# B&R Automation Studio project perfxxl (part 3)

#### sram.c
```c
#ifdef _DEFAULT_INCLUDES
	#include <AsDefault.h>
#endif
/****************************************************************************/
/*	Zugriff auf remanenten Speicher*/
/*																			*/
/*																			*/
/*	Versionsgeschichte:														*/
/*  Version		Datum		Änderung										von		*/
/*	1.00		16.09.02	erste Implementation								HA		*/
/*	1.10		31.03.03	bei Änderung Aufl. und Speed speichern		HA		*/
/*	1.11		20.05.03	floats auf Gültigkeit prüfen				HA		*/
/*																			*/
/****************************************************************************/

#include <bur/plc.h>
#include <bur/plctypes.h>
#include <math.h>
#include <asstring.h>
#include "glob_var.h"
#include "egmglob_var.h"
#include <fileio.h>

#define	MAXFILELIST	32
#define MAXFILES	50
#define MAXFILENAMELENGTH	32

#define OVERALLSRAMSIZEWORDS 12500
#define OVERALLSRAMSIZEEBYTES 25000

typedef struct{
BOOL enable;
UDINT len;
UDINT offset;
UDINT	address;
}puttyp;
typedef struct{
BOOL enable;
UDINT len;
UDINT offset;
UDINT	address;
}gettyp;
puttyp put;
gettyp get;

_LOCAL UINT             wStatus, wError;
_LOCAL UDINT            dwDirNum, dwFileNum, dwCounter;
_LOCAL DirInfo_typ      DInfo;
_LOCAL DirCreate_typ      DCreate;
_LOCAL BOOL Created;
_GLOBAL BOOL PreheatParamEnter,DeveloperTankParamEnter;

_LOCAL STRING targetstring[20];
int i,j;
USINT tmp[OVERALLSRAMSIZEEBYTES];
_GLOBAL USINT *TmpPtr;

int len;
_GLOBAL UDINT	PlatesMade;
_GLOBAL	BOOL	savePlatesMade;
		BOOL	loadPlatesMade;
_GLOBAL	STRING FileIOName[MAXFILENAMELENGTH];
_GLOBAL	STRING	FileType[5];
_GLOBAL	UDINT *FileIOData;
_GLOBAL	UDINT	FileIOLength;
_GLOBAL	BOOL	WriteFileCmd,ReadFileCmd,DeleteFileCmd,WriteFileOK,ReadFileOK,DeleteFileOK,
				FileNotExisting,ReadDirCmd,ReadDirOK,NoDisk;
_GLOBAL	BOOL ParameterChanged;

_LOCAL	BOOL	StartUp,ReadActive,WriteActive,SaveToFile;
_LOCAL	BOOL	ClearSRAM,LoadSRAMFromFile;
_GLOBAL BOOL	PutTmpDataToSRAM,GetTmpDataFromSRAM;
BOOL	DontResetMotorData;
_GLOBAL BOOL MirroredMachine;

_GLOBAL SINT SRAM[OVERALLSRAMSIZEEBYTES]	_VAR_RETAIN;
_GLOBAL BOOL	EGMsaveParameterData;
_LOCAL INT	Test1,Test2,Test3;

_LOCAL	STRING	MagicNumber[10];
_GLOBAL	DATE_AND_TIME	OffTime,OnTime;

void SRAMPut(puttyp *param)
{
	memcpy(&SRAM[0]+param->offset*2,(SINT *)(param->address),param->len *2);
}

void SRAMGet(gettyp *param)
{
	memcpy((SINT *)(param->address),&SRAM[0]+param->offset*2,param->len *2);
}

void InitXData(void)
{
	ClearSRAM = 0;
	X_Param.RefSpeed1		= 20;
	X_Param.RefSpeed2		= 10;
	X_Param.RefSpeed3		= 5;
	X_Param.ManSpeed1		= 20;
	X_Param.ManSpeed2		= 50;
	X_Param.ParkSpeed		= 195;
/*Positionen*/
	X_Param.Offset			= 0;		/*Nullpunktkorrektur*/
	X_Param.ParkPosition	= -3.0;
	X_Param.InkrementeProMm	= 2730.666;
	X_Param.MinPosition	= -37.0;
	X_Param.MaxPosition	= 1258.0;
}

void InitGlobalData(void)
{
	PlatesMade = 0;

	PlateParameter.XOffset = 0.0;
	PlateParameter.YOffset = 0.0;
	PlateParameter.Length  = 320.0;
	PlateParameter.Width   = 600.0;
	PlateParameter.Thickness = 0.30;
	PlateParameter.Sensitivity = 100.0;

	strcpy(GlobalParameter.MachineName,"LS Performance XXL");
	strcpy(GlobalParameter.MachineNumber,"12345");
	strcpy(GlobalParameter.CustomerName,"eintragen!!");
	GlobalParameter.ScansPerMinute			= 96000;
	GlobalParameter.Resolution				= 1270;
	GlobalParameter.MaxPlateLength			= 1250; /*not in use*/
	GlobalParameter.MinPlateLength			= 250;  /*not in use*/
	GlobalParameter.TrolleyRightOffset		= 73650;/*not in use*/
	GlobalParameter.AlternatingTrolleys		= FALSE;/*not in use*/
	GlobalParameter.XSimulation				= FALSE;
	GlobalParameter.TBSimulation			= FALSE;
	GlobalParameter.ProcessorSimulation		= FALSE;
	GlobalParameter.PunchSimulation			= FALSE;
	GlobalParameter.PaperRemoveEnabled		= TRUE;
	GlobalParameter.UseOldTiffBlaster		= FALSE;/*not in use*/
	GlobalParameter.Dummy					= FALSE;
	GlobalParameter.Language				= 1;
	GlobalParameter.DeloaderTurnStation		= 0;
	GlobalParameter.FlexibleFeeder			= 0;
	GlobalParameter.AutomaticTrolleyOpenClose	= TRUE;
	GlobalParameter.TrolleyLeft				= 0;
	GlobalParameter.TrolleyRight			= 0;
	GlobalParameter.RealLaserPower			= 300;
	GlobalParameter.LaserPower = (GlobalParameter.RealLaserPower+5) / 10;
	GlobalParameter.MirroredMachine			= 0; /* !=42: not mirrored; 42: mirrored*/
	GlobalParameter.SlowModeWaitTime		= 2000; /* 20 sec default */
	GlobalParameter.DisableSlowMode			= 1;

	Expose_Param.ScansPerMinute			= 96000;
	Expose_Param.Resolution				= 1270;

/*TROLLEYS*/
	for(i = 0; i < MAXTROLLEYS; i++)
	{
		strcpy( Trolleys[i].Name,"Trolley");
		Trolleys[i].Number 				= i;	/*bugfix i instead of i+1*/
		Trolleys[i].PlateType 			= 1;
		Trolleys[i].Empty 				= FALSE;
		Trolleys[i].Single 				= FALSE;
		Trolleys[i].Double 				= TRUE;
		Trolleys[i].NoCover		 		= FALSE;
		Trolleys[i].LeftStack 			= TRUE;
		Trolleys[i].RightStack 			= FALSE;
		Trolleys[i].PlatesLeft 			= 0;
		Trolleys[i].PlatesRight 		= 0;
		Trolleys[i].OpenStart 			= 175600;
		Trolleys[i].OpenStop 			= 353100;
		Trolleys[i].CloseStart 			= 353100;
		Trolleys[i].CloseStop 			= 174440;
		Trolleys[i].TakePlateLeft 		= 8300;  /* not in use*/
		Trolleys[i].TakePlateRight 		= 57000; /* not in use*/
		Trolleys[i].TakePaperLeft 		= 335000;
		Trolleys[i].TakePaperRight 		= 335000;
		Trolleys[i].EmptyLeft 			= FALSE;
		Trolleys[i].EmptyRight 			= FALSE;
		Trolleys[i].EmptyPositions[0] 			= 64000;
		Trolleys[i].EmptyPositions[1] 			= 64000;
		Trolleys[i].EmptyPositions[2] 			= 64000;
	}

/*PLATETYPES*/
	for(i = 0; i < MAXPLATETYPES; i++)
	{
		strcpy( PlateTypes[i].Name,"Platte");
		PlateTypes[i].Number 				= i; /*bugfix i instead of i+1*/
		PlateTypes[i].Length 				= 312.00;
		PlateTypes[i].XOffset 				= 0.00;
		PlateTypes[i].Width 				= 600.00;
		PlateTypes[i].YOffset 				= 10.00;
		PlateTypes[i].Thickness 				= 0.32;
		PlateTypes[i].TakePlatePosition 				= 100000;
		PlateTypes[i].ReleasePlatePosition 			= 10000;
		PlateTypes[i].ReleasePlatePosition2 			= 10000;
		PlateTypes[i].TurnMode							= 0;
		PlateTypes[i].SeparateBeltTracks	= 0;
	}

/*FEEDER*/
	FeederParameter.HorizontalPositions.ReleasePlate 				= 500;/* not in use*/
	FeederParameter.HorizontalPositions.TakePlate 				= 1500;/* not in use*/
	FeederParameter.VerticalPositions.Up 							= 2000;
	FeederParameter.VerticalPositions.EnablePaperRemove 		= 22000;
	FeederParameter.VerticalPositions.AboveTrolley 				= 22000;
	FeederParameter.VerticalPositions.MaxDown	 				= 70000;
	FeederParameter.VerticalPositions.PreRelease 					= 2000;
	FeederParameter.VerticalPositions.ReleasePlate 				= 2000;
	FeederParameter.VerticalPositions.SpeedChangePosition 		= 18200;
	FeederParameter.VacuumOnTime								= 100;
	FeederParameter.VacuumOffTime								= 50;
	FeederParameter.SpeedUpSlow									= 700;
	FeederParameter.SpeedUpFast									= 7000;
	FeederParameter.Stack0Pos									= -186000;/* not in use*/
	FeederParameter.Stack20Pos									= -183248;/* not in use*/
	FeederParameter.SlowDownPos									= 1000;
	FeederParameter.StackDetectSpeed							= 500;
	FeederParameter.PanoramaAdapter							= 25000;
	FeederParameter.SuckRepitions								= 0;
	FeederParameter.ShakeRepitions								= 0;
	FeederParameter.ShakeTime									= 30;
	FeederParameter.ShakeWay									= 3000;
	FeederParameter.WaitForExposer								= 0;
	FeederParameter.IgnoreVacuumSwitch							= 0;
	FeederParameter.HorPositionPano							= 2000;
	FeederParameter.MaxTablePosition							= 170.0;
	FeederParameter.MinTablePosDrop							= 1180.0;
	FeederParameter.DropOffset									= 20.0;/* not in use */

/* Paper Remove */
	PaperRemoveParameter.HorizontalPositions.EnableFeeder 			= 126000;
	PaperRemoveParameter.HorizontalPositions.PaperReleaseSingle		= 70000;
	PaperRemoveParameter.HorizontalPositions.PaperReleasePanorama	= 50000;

/*folgende Werte werden im Ablauf errechnet*/
	PaperRemoveParameter.HorizontalPositions.PaperRemoveLeft		= -120000;
	PaperRemoveParameter.HorizontalPositions.PaperRemoveRight		= -196000;
	PaperRemoveParameter.HorizontalPositions.TrolleyCloseRightStart	= -196000;
	PaperRemoveParameter.HorizontalPositions.TrolleyCloseRightStop	= -178000;
	PaperRemoveParameter.HorizontalPositions.TrolleyOpenRightStart	= -178000;
	PaperRemoveParameter.HorizontalPositions.TrolleyOpenRightStop	= -196000;
	PaperRemoveParameter.HorizontalPositions.PaletteDetectStartPos	=  120000;
	PaperRemoveParameter.HorizontalPositions.PaletteDetectEndPos	=  130000;
	PaperRemoveParameter.HorizontalPositions.TrolleyOpenRightStop	= -196000;
/* bis hier*/
	PaperRemoveParameter.VerticalPositions.Up						= 300;
	PaperRemoveParameter.VerticalPositions.Down						= 13000;
	PaperRemoveParameter.VerticalPositions.OnTrolley				= 1200;
	PaperRemoveParameter.TrolleyOpenCloseSpeed						= 1000;
	PaperRemoveParameter.PaperRemoveSpeed							= 5000;
	PaperRemoveParameter.TrolleyDetectSpeed							= 500;
	PaperRemoveParameter.TrolleyOpenDownSpeed						= 300;
	PaperRemoveParameter.TrolleyOpenUpSpeed							= 800;
	PaperRemoveParameter.PaperRemoveDownSpeed						= 1000;
	PaperRemoveParameter.PaperRemoveUpSpeed							= 1500;
	PaperRemoveParameter.TrolleyDetectStartPos						= 180000;
	PaperRemoveParameter.TrolleyDetectEndPos						= 280000;
	PaperRemoveParameter.MaxCurrentDown								= 2000;
	PaperRemoveParameter.MaxCurrentUp								= 5000;
	PaperRemoveParameter.GripOnTime									= 100;
	PaperRemoveParameter.GripOffTime								= 80;
	PaperRemoveParameter.TimeoutOnTrolley							= 100;
	PaperRemoveParameter.PaletteDetectSpeed							= 300;
	PaperRemoveParameter.TimeoutUpFromTrolley						= 100;
	PaperRemoveParameter.TimeoutOpenTrolleySmall					= 1000;/* not in use*/
	PaperRemoveParameter.TimeoutOpenTrolleyBig						= 2000;/* not in use*/
	PaperRemoveParameter.PaperGripCycles							= 0;
	PaperRemoveParameter.HorPositionPano							= 300000;
	PaperRemoveParameter.PaperReleasePosVertical					= 10000;

/*Adjuster*/
	AdjusterParameter.PinsUpTime									= 20;
	AdjusterParameter.PinsDownTime									= 20;
	AdjusterParameter.TableVacuumOnDelay							= 10;
	AdjusterParameter.TableVacuumOffDelay							= 20;
	AdjusterParameter.AdjVacuumOnDelay							= 50;
	AdjusterParameter.AdjVacuumOffDelay							= 10;
	AdjusterParameter.BlowairOnDelay								= 10;
	AdjusterParameter.BlowairOffDelay								= 10;
	AdjusterParameter.TimeoutAdjustedPosition						= 100;
	AdjusterParameter.MaxFailedPlates								= 0;
	AdjusterParameter.AddBlowairValveDelay						    = 1;
	AdjusterParameter.MaxAttempts									= 3;
	AdjusterParameter.AdjActiveTime									= 30;
	AdjusterParameter.AdjInactiveTime								= 30;
	AdjusterParameter.AdjustSim										= FALSE;
	AdjusterParameter.FeederAdjustposition							= 6450;
	AdjusterParameter.FeederFixposition							    = 7500;

/*DELOADER*/
	DeloaderParameter.MaxPlateTakePosition							= 100000;
	DeloaderParameter.PlateReleasePosition							= 10000;
	DeloaderParameter.PlateReleasePosition2							= 10000;
	DeloaderParameter.TurnEnabledPosition							= 50000;
	DeloaderParameter.MinTablePositionTake							= 235.0;
	DeloaderParameter.MaxTablePositionRelease						= 500.0;
	DeloaderParameter.Turn0Position									= 15400;
	DeloaderParameter.Turn90Position								= 26100;
	DeloaderParameter.Turn180Position								= 36800;
	DeloaderParameter.ConveyorBeltSpeed								= 300;
	DeloaderParameter.TableDeloadSpeedManual								= 200.0;
	DeloaderParameter.TableDeloadSpeed								= 200.0;
	DeloaderParameter.TurnSpeed										= 2000;
	DeloaderParameter.VacuumOnTime									= 50;
	DeloaderParameter.VacuumOffTime									= 50;
	DeloaderParameter.PlateLengthAddition								= 120;
	DeloaderParameter.ConveyorBeltDelay								= 500;
	DeloaderParameter.EGMStopDelay									= 4500;
	DeloaderParameter.ShiftedLayingOff								= 0;
	DeloaderParameter.PinsUpDelay									= 200;
	DeloaderParameter.PinsDownDelay								= 200;
	DeloaderParameter.EnableStopPins								= 0;
	DeloaderParameter.SeparateSensors								= 0;
	DeloaderParameter.StartTablePosition                           = -6.0;
	DeloaderParameter.EndTablePosition                             = 1258;
	DeloaderParameter.ConvLateralMoveTime                          = 200;
	DeloaderParameter.ConvLateralPulseTime                          = 30;

	for (i=1;i<MAXLASERPOWERSETTINGS;i++)
	{
		LaserPowerSettings[i].Resolution = 0;
		for (j = 1;j<MAXPLATETYPES;j++)
			LaserPowerSettings[i].LaserPower[j] = 0;
	}
}

void InitMotorData(void)
{
	Motors[FEEDER_VERTICAL].Parameter.ControllerIFact						= 20;
	strcpy(Motors[FEEDER_VERTICAL].Parameter.Function,"Feeder vertical");
	Motors[FEEDER_VERTICAL].Parameter.Priority						= 1;
	Motors[FEEDER_VERTICAL].Parameter.IncrementsPerMm				= 140;
	Motors[FEEDER_VERTICAL].Parameter.ReferenceSpeed				= 500;
	Motors[FEEDER_VERTICAL].Parameter.ReferenceDirectionNegative	= 0;
	Motors[FEEDER_VERTICAL].Parameter.ReferencePeekCurrent			= 3000;
	Motors[FEEDER_VERTICAL].Parameter.DefaultPeekCurrent			= 8000;
	Motors[FEEDER_VERTICAL].Parameter.ReferenceContCurrent			= 2500;
	Motors[FEEDER_VERTICAL].Parameter.DefaultContCurrent			= 2000;
	Motors[FEEDER_VERTICAL].Parameter.ReferencePropFact				= 2;
	Motors[FEEDER_VERTICAL].Parameter.DefaultPropFact				= 8;
	Motors[FEEDER_VERTICAL].Parameter.ReferenceOffset				= 2000;
	Motors[FEEDER_VERTICAL].Parameter.ReferenceAcceleration			= 50;
	Motors[FEEDER_VERTICAL].Parameter.DefaultAcceleration			= 300;
	Motors[FEEDER_VERTICAL].Parameter.ManSpeed						= 500;
	Motors[FEEDER_VERTICAL].Parameter.MaximumSpeed					= 10000;
	Motors[FEEDER_VERTICAL].Parameter.MaximumPosition				= 70000;
	Motors[FEEDER_VERTICAL].Parameter.MinimumPosition				= 100;
	Motors[FEEDER_VERTICAL].Parameter.PositionWindow				= 200;

	Motors[FEEDER_HORIZONTAL].Parameter.ControllerIFact						= 20;
	strcpy(Motors[FEEDER_HORIZONTAL].Parameter.Function,"Feeder horizontal");
	Motors[FEEDER_HORIZONTAL].Parameter.Priority					= 1;
	Motors[FEEDER_HORIZONTAL].Parameter.IncrementsPerMm				= 140;
	Motors[FEEDER_HORIZONTAL].Parameter.ReferenceSpeed				= 500;
	Motors[FEEDER_HORIZONTAL].Parameter.ReferenceDirectionNegative	= 1;
	Motors[FEEDER_HORIZONTAL].Parameter.ReferencePeekCurrent		= 3000;
	Motors[FEEDER_HORIZONTAL].Parameter.DefaultPeekCurrent			= 8000;
	Motors[FEEDER_HORIZONTAL].Parameter.ReferenceContCurrent		= 2500;
	Motors[FEEDER_HORIZONTAL].Parameter.DefaultContCurrent			= 6000;
	Motors[FEEDER_HORIZONTAL].Parameter.ReferencePropFact			= 2;
	Motors[FEEDER_HORIZONTAL].Parameter.DefaultPropFact				= 8;
	Motors[FEEDER_HORIZONTAL].Parameter.ReferenceOffset				= 2000;
	Motors[FEEDER_HORIZONTAL].Parameter.ReferenceAcceleration		= 50;
	Motors[FEEDER_HORIZONTAL].Parameter.DefaultAcceleration			= 300;
	Motors[FEEDER_HORIZONTAL].Parameter.ManSpeed					= 500;
	Motors[FEEDER_HORIZONTAL].Parameter.MaximumSpeed				= 10000;
	Motors[FEEDER_HORIZONTAL].Parameter.MaximumPosition				= 100000;
	Motors[FEEDER_HORIZONTAL].Parameter.MinimumPosition				= 100;
	Motors[FEEDER_HORIZONTAL].Parameter.PositionWindow				= 100;

	Motors[PAPERREMOVE_HORIZONTAL].Parameter.ControllerIFact					= 20;
	strcpy(Motors[PAPERREMOVE_HORIZONTAL].Parameter.Function,"Papierentf. horiz.");
	Motors[PAPERREMOVE_HORIZONTAL].Parameter.Priority				= 1;
	Motors[PAPERREMOVE_HORIZONTAL].Parameter.IncrementsPerMm		= 140;
	Motors[PAPERREMOVE_HORIZONTAL].Parameter.ReferenceSpeed			= 500;
	Motors[PAPERREMOVE_HORIZONTAL].Parameter.ReferenceDirectionNegative	= 0;
	Motors[PAPERREMOVE_HORIZONTAL].Parameter.ReferencePeekCurrent	= 6000;
	Motors[PAPERREMOVE_HORIZONTAL].Parameter.DefaultPeekCurrent		= 8000;
	Motors[PAPERREMOVE_HORIZONTAL].Parameter.ReferenceContCurrent	= 4000;
	Motors[PAPERREMOVE_HORIZONTAL].Parameter.DefaultContCurrent		= 6000;
	Motors[PAPERREMOVE_HORIZONTAL].Parameter.ReferencePropFact		= 6;
	Motors[PAPERREMOVE_HORIZONTAL].Parameter.DefaultPropFact		= 8;
	Motors[PAPERREMOVE_HORIZONTAL].Parameter.ReferenceOffset		= 126000;
	Motors[PAPERREMOVE_HORIZONTAL].Parameter.ReferenceAcceleration	= 50;
	Motors[PAPERREMOVE_HORIZONTAL].Parameter.DefaultAcceleration	= 300;
	Motors[PAPERREMOVE_HORIZONTAL].Parameter.ManSpeed				= 500;
	Motors[PAPERREMOVE_HORIZONTAL].Parameter.MaximumSpeed			= 10000;
	Motors[PAPERREMOVE_HORIZONTAL].Parameter.MaximumPosition		= 360000;
	Motors[PAPERREMOVE_HORIZONTAL].Parameter.MinimumPosition		= 500;
	Motors[PAPERREMOVE_HORIZONTAL].Parameter.PositionWindow			= 1000;

	Motors[PAPERREMOVE_VERTICAL].Parameter.ControllerIFact					= 20;
	strcpy(Motors[PAPERREMOVE_VERTICAL].Parameter.Function,"Papierentf. vertik.");
	Motors[PAPERREMOVE_VERTICAL].Parameter.Priority					= 1;
	Motors[PAPERREMOVE_VERTICAL].Parameter.IncrementsPerMm			= 140;
	Motors[PAPERREMOVE_VERTICAL].Parameter.ReferenceSpeed			= 200;
	Motors[PAPERREMOVE_VERTICAL].Parameter.ReferenceDirectionNegative	= 1;
	Motors[PAPERREMOVE_VERTICAL].Parameter.ReferencePeekCurrent		= 6000;
	Motors[PAPERREMOVE_VERTICAL].Parameter.DefaultPeekCurrent		= 8000;
	Motors[PAPERREMOVE_VERTICAL].Parameter.ReferenceContCurrent		= 4500;
	Motors[PAPERREMOVE_VERTICAL].Parameter.DefaultContCurrent		= 4000;
	Motors[PAPERREMOVE_VERTICAL].Parameter.ReferencePropFact		= 2;
	Motors[PAPERREMOVE_VERTICAL].Parameter.DefaultPropFact			= 8;
	Motors[PAPERREMOVE_VERTICAL].Parameter.ReferenceOffset			= 300;
	Motors[PAPERREMOVE_VERTICAL].Parameter.ReferenceAcceleration	= 50;
	Motors[PAPERREMOVE_VERTICAL].Parameter.DefaultAcceleration		= 300;
	Motors[PAPERREMOVE_VERTICAL].Parameter.ManSpeed					= 500;
	Motors[PAPERREMOVE_VERTICAL].Parameter.MaximumSpeed				= 1000;
	Motors[PAPERREMOVE_VERTICAL].Parameter.MaximumPosition			= 13000;
	Motors[PAPERREMOVE_VERTICAL].Parameter.MinimumPosition			= 100;
	Motors[PAPERREMOVE_VERTICAL].Parameter.PositionWindow			= 30;

	memcpy(&Motors[PAPERREMOVE_VERTICAL2],&Motors[PAPERREMOVE_VERTICAL],sizeof(Motors[PAPERREMOVE_VERTICAL]));
	strcpy(Motors[PAPERREMOVE_VERTICAL].Parameter.Function,"Papierentf. vertik. 2");

	Motors[ADJUSTER].Parameter.ControllerIFact								= 20;
	strcpy(Motors[ADJUSTER].Parameter.Function,"Ausrichtband");
	Motors[ADJUSTER].Parameter.Priority								= 1;
	Motors[ADJUSTER].Parameter.IncrementsPerMm						= 96;
	Motors[ADJUSTER].Parameter.ReferenceSpeed						= 500;
	Motors[ADJUSTER].Parameter.ReferenceDirectionNegative			= 1;
	Motors[ADJUSTER].Parameter.ReferencePeekCurrent					= 3000;
	Motors[ADJUSTER].Parameter.DefaultPeekCurrent					= 8000;
	Motors[ADJUSTER].Parameter.ReferenceContCurrent					= 2500;
	Motors[ADJUSTER].Parameter.DefaultContCurrent					= 6000;
	Motors[ADJUSTER].Parameter.ReferencePropFact					= 2;
	Motors[ADJUSTER].Parameter.DefaultPropFact						= 8;
	Motors[ADJUSTER].Parameter.ReferenceOffset						= 2000;
	Motors[ADJUSTER].Parameter.ReferenceAcceleration				= 50;
	Motors[ADJUSTER].Parameter.DefaultAcceleration					= 200;
	Motors[ADJUSTER].Parameter.ManSpeed								= 500;
	Motors[ADJUSTER].Parameter.MaximumSpeed							= 10000;
	Motors[ADJUSTER].Parameter.MaximumPosition						= 99999999;
	Motors[ADJUSTER].Parameter.MinimumPosition						= -99999999;
	Motors[ADJUSTER].Parameter.PositionWindow						= 100;

	Motors[DELOADER_TURN].Parameter.ControllerIFact					= 2;
	strcpy(Motors[DELOADER_TURN].Parameter.Function,"Entlader Rot.");
	Motors[DELOADER_TURN].Parameter.Priority						= 1;
	Motors[DELOADER_TURN].Parameter.IncrementsPerMm					= 200;
	Motors[DELOADER_TURN].Parameter.ReferenceSpeed					= 250;
	Motors[DELOADER_TURN].Parameter.ReferenceDirectionNegative		= 1;
	Motors[DELOADER_TURN].Parameter.ReferencePeekCurrent			= 3000;
	Motors[DELOADER_TURN].Parameter.DefaultPeekCurrent				= 8000;
	Motors[DELOADER_TURN].Parameter.ReferenceContCurrent			= 2500;
	Motors[DELOADER_TURN].Parameter.DefaultContCurrent				= 3000;
	Motors[DELOADER_TURN].Parameter.ReferencePropFact				= 4;
	Motors[DELOADER_TURN].Parameter.DefaultPropFact					= 8;
	Motors[DELOADER_TURN].Parameter.ReferenceOffset					= 14800;
	Motors[DELOADER_TURN].Parameter.ReferenceAcceleration			= 50;
	Motors[DELOADER_TURN].Parameter.DefaultAcceleration				= 100;
	Motors[DELOADER_TURN].Parameter.ManSpeed						= 100;
	Motors[DELOADER_TURN].Parameter.MaximumSpeed					= 700;
	Motors[DELOADER_TURN].Parameter.MaximumPosition					= 50000;
	Motors[DELOADER_TURN].Parameter.MinimumPosition					= 100;
	Motors[DELOADER_TURN].Parameter.PositionWindow					= 50;

	Motors[DELOADER_HORIZONTAL].Parameter.ControllerIFact					= 20;
	strcpy(Motors[DELOADER_HORIZONTAL].Parameter.Function,"Entlader horiz.");
	Motors[DELOADER_HORIZONTAL].Parameter.Priority					= 1;
	Motors[DELOADER_HORIZONTAL].Parameter.IncrementsPerMm			= 140;
	Motors[DELOADER_HORIZONTAL].Parameter.ReferenceSpeed			= 500;
	Motors[DELOADER_HORIZONTAL].Parameter.ReferenceDirectionNegative	= 1;
	Motors[DELOADER_HORIZONTAL].Parameter.ReferencePeekCurrent		= 3000;
	Motors[DELOADER_HORIZONTAL].Parameter.DefaultPeekCurrent		= 8000;
	Motors[DELOADER_HORIZONTAL].Parameter.ReferenceContCurrent		= 2500;
	Motors[DELOADER_HORIZONTAL].Parameter.DefaultContCurrent		= 4000;
	Motors[DELOADER_HORIZONTAL].Parameter.ReferencePropFact			= 2;
	Motors[DELOADER_HORIZONTAL].Parameter.DefaultPropFact			= 8;
	Motors[DELOADER_HORIZONTAL].Parameter.ReferenceOffset			= 50000;
	Motors[DELOADER_HORIZONTAL].Parameter.ReferenceAcceleration		= 50;
	Motors[DELOADER_HORIZONTAL].Parameter.DefaultAcceleration		= 300;
	Motors[DELOADER_HORIZONTAL].Parameter.ManSpeed					= 500;
	Motors[DELOADER_HORIZONTAL].Parameter.MaximumSpeed				= 5000;
	Motors[DELOADER_HORIZONTAL].Parameter.MaximumPosition			= 110000;
	Motors[DELOADER_HORIZONTAL].Parameter.MinimumPosition			= 100;
	Motors[DELOADER_HORIZONTAL].Parameter.PositionWindow			= 200;

	Motors[CONVEYORBELT].Parameter.ControllerIFact							= 20;
	strcpy(Motors[CONVEYORBELT].Parameter.Function,"Auslaufband");
	Motors[CONVEYORBELT].Parameter.Priority							= 1;
	Motors[CONVEYORBELT].Parameter.IncrementsPerMm					= 100;
	Motors[CONVEYORBELT].Parameter.ReferenceSpeed					= 500;
	Motors[CONVEYORBELT].Parameter.ReferenceDirectionNegative		= 1;
	Motors[CONVEYORBELT].Parameter.ReferencePeekCurrent				= 3000;
	Motors[CONVEYORBELT].Parameter.DefaultPeekCurrent				= 8000;
	Motors[CONVEYORBELT].Parameter.ReferenceContCurrent				= 2500;
	Motors[CONVEYORBELT].Parameter.DefaultContCurrent				= 3000;
	Motors[CONVEYORBELT].Parameter.ReferencePropFact				= 2;
	Motors[CONVEYORBELT].Parameter.DefaultPropFact					= 8;
	Motors[CONVEYORBELT].Parameter.ReferenceOffset					= 500;
	Motors[CONVEYORBELT].Parameter.ReferenceAcceleration			= 50;
	Motors[CONVEYORBELT].Parameter.DefaultAcceleration				= 100;
	Motors[CONVEYORBELT].Parameter.ManSpeed							= 500;
	Motors[CONVEYORBELT].Parameter.MaximumSpeed						= 1000;
	Motors[CONVEYORBELT].Parameter.MaximumPosition					= 99999999;
	Motors[CONVEYORBELT].Parameter.MinimumPosition					= -99999999;
	Motors[CONVEYORBELT].Parameter.PositionWindow					= 50;
}

/**********************************************************************************/
/**********************************************************************************/
/**********************************************************************************/
void EGMSetDefaults(void)
{
	int i;
	char tmpstr[5];

/* Globals*/
	strcpy(EGMGlobalParam.Version,gVERSION);
	EGMGlobalParam.MachineType =						BLUEFIN_XS;
	MachineType = EGMGlobalParam.MachineType;
	EGMGlobalParam.Unit_Rpm = 							1;
	EGMGlobalParam.Unit_Propulsion = 					1;
	EGMGlobalParam.Unit_Temperature = 					1;
	EGMGlobalParam.Unit_Length = 						0;
	EGMGlobalParam.Unit_Area = 							0;
	EGMGlobalParam.Unit_Volume = 						0;
	EGMGlobalParam.MainMotorFactor = 					3.0/32767.0;
	EGMGlobalParam.MaxPlateSizeX = 						1050;
	EGMGlobalParam.MaxPlateSizeY = 						650;
	EGMGlobalParam.BrushFactor =                        230.0/32767.0;
	EGMGlobalParam.UseGumFlowControl =					0;
	EGMGlobalParam.UseDevCircFlowControl =				0;
	EGMGlobalParam.UsePrewashFlowControl = 				0;
	EGMGlobalParam.UseRinseFlowControl = 				0;
	EGMGlobalParam.UseTopUpFlowControl = 				0;
	EGMGlobalParam.UseReplFlowControl = 				0;
	EGMGlobalParam.PlateDirection = 					0;	/* 0=right to left, 1=left to right */
	EGMGlobalParam.DeveloperPulsesPerLiter =			1200;
	EGMGlobalParam.ReplenisherPulsesPerLiter =			1200;
	EGMGlobalParam.GumPulsesPerLiter =					1200;
	EGMGlobalParam.ScreensaverTime =					300; /* in sec -> 5 min*/

/* Main Motor*/
	EGMMainMotor.Auto = 0;
	EGMMainMotor.Manual = 1;
	EGMMainMotor.Start = 0;
	EGMMainMotor.Stop = 0;
	EGMMainMotor.Enable = 0;
	EGMMainMotor.RatedRpm = 0;
	EGMMainMotor.AutoRatedRpm = 0;
	EGMMainMotor.RealRpm = 0;

/* brush Motor*/
	EGMBrushMotor.Auto = 0;
	EGMBrushMotor.Manual = 1;
	EGMBrushMotor.Start = 0;
	EGMBrushMotor.Stop = 0;
	EGMBrushMotor.Enable = 0;
	EGMBrushMotor.RatedRpm = 0;
	EGMBrushMotor.AutoRatedRpm = 0;
	EGMBrushMotor.RealRpm = 0;

/* Automatik*/
	EGMAutoParam.Speed =					19338;
	EGMAutoParam.BrushSpeed =				25700;
	EGMAutoParam.PreheatTemp = 				1600;
	EGMAutoParam.PreheatTemp2 = 			1600;
	EGMAutoParam.DeveloperTemp = 			230;
	EGMAutoParam.StandbyDelay =				3000;
	EGMAutoParam.StandbySpeed =			8595;
	EGMAutoParam.MaxPlateSizeX =			1050;
	EGMAutoParam.MaxPlateSizeY =			650;
	EGMAutoParam.StandbyBrushSpeed =		5507;
	EGMAutoParam.WaitGumBackTime = 		120;
	EGMAutoParam.GumRinsingTime = 			120;
	EGMAutoParam.WaitGumRinseTime = 		50;

/* Preheat*/
	for (i=0;i<4;i++)
	{
		EGMPreheatParam.RatedTemp[i] = 				1600;
		EGMPreheatParam.RatedTempCorr[i] =			1600;
		EGMPreheatParam.ReglerParam[i].Kp =			3.8;
		EGMPreheatParam.ReglerParam[i].Tn =			48000.0;
		EGMPreheatParam.ReglerParam[i].Tv =			12000.0;
		EGMPreheatParam.ReglerParam[i].Tf =			1200.0;
		EGMPreheatParam.ReglerParam[i].Kw =			1.0;
		EGMPreheatParam.ReglerParam[i].Kfbk =		1.0;
		EGMPreheatParam.ReglerParam[i].d_mode =	1;
		EGMPreheatParam.ReglerParam[i].tminpuls =	10;
		EGMPreheatParam.ReglerParam[i].tperiod =		200;
		EGMPreheatParam.ReglerParam[i].SetpointTracking =	1;

		EGMPreheatParam.EndSetpoint[i] =				1600;
		EGMPreheatParam.StartOverheat[i] =			750;
		EGMPreheatParam.StartAmbient[i] =			300;
		EGMPreheatParam.EndAmbient[i] =				940;
	}

	EGMPreheatParam.ToleratedDevPos =			30;
	EGMPreheatParam.ToleratedDevNeg =			30;
	EGMPreheatParam.MaxOKTemp =				1630;
	EGMPreheatParam.MinOKTemp =				1570;
	EGMPreheatParam.SetPointCorrTMin=			30;
	EGMPreheatParam.SetPointCorrMax=			500;

/* Entwickler*/
	EGMDeveloperTankParam.RatedTemp =				230;
	EGMDeveloperTankParam.TempOffset =				-17;
	EGMDeveloperTankParam.ToleratedDevPos =			10;
	EGMDeveloperTankParam.ToleratedDevNeg =			10;
	EGMDeveloperTankParam.CoolingOnY =					-15;
	EGMDeveloperTankParam.MaxOKTemp =				240;
	EGMDeveloperTankParam.MinOKTemp =				220;
	EGMDeveloperTankParam.MinOnTimeCooling =			700;

	EGMDeveloperTankParam.StartRefillDelay =				0;
	EGMDeveloperTankParam.StopRefillDelay =				0;

	EGMDeveloperTankParam.ReglerParam.Kp =			10.0;
	EGMDeveloperTankParam.ReglerParam.Tn =			0.0;
	EGMDeveloperTankParam.ReglerParam.Tv =			400.0;
	EGMDeveloperTankParam.ReglerParam.Tf =				100.0;
	EGMDeveloperTankParam.ReglerParam.Kw =			1.0;
	EGMDeveloperTankParam.ReglerParam.Kfbk =			1.0;
	EGMDeveloperTankParam.ReglerParam.d_mode =		1;
	EGMDeveloperTankParam.ReglerParam.tminpuls =		1;
	EGMDeveloperTankParam.ReglerParam.tperiod =		20;
	EGMDeveloperTankParam.ReglerParam.SetpointTracking =	0;

	EGMDeveloperTankParam.ReplenishingMode =			1;
	EGMDeveloperTankParam.EnableStandbyReplenishing =	1;
	EGMDeveloperTankParam.EnableOffReplenishing =		0;
	EGMDeveloperTankParam.TopUpMode =						1;
	EGMDeveloperTankParam.ReplenishmentPerSqm =		100.0;
	EGMDeveloperTankParam.ReplenishmentPerPlate =		20.0;
	EGMDeveloperTankParam.StandbyReplenishment =		50.0;
	EGMDeveloperTankParam.OffReplenishment =			20.0;
	EGMDeveloperTankParam.StandbyReplenishmentIntervall = 90;
	EGMDeveloperTankParam.PumpMlPerSec =				30.0;
	EGMDeveloperTankParam.MinPumpOnTime =			300;
	EGMDeveloperTankParam.MinPumpOnTimeStandby =	300;

	EGMDeveloperTankParam.TopUpMode =				1;
	EGMDeveloperTankParam.TopUpPerSqm =				50.0;
	EGMDeveloperTankParam.TopUpPerPlate =			20.0;
	EGMDeveloperTankParam.TopUpPumpMlPerSec =		30.0;
	EGMDeveloperTankParam.TopUpMinPumpOnTime =		300;

/* PreWash*/
	EGMPrewashParam.ReplenishingMode =				1;
	EGMPrewashParam.ReplenishmentPerSqm =			1000.0;
	EGMPrewashParam.ReplenishmentPerPlate = 			300.0;
	EGMPrewashParam.ReplenishmentIntervall = 			0;
	EGMPrewashParam.PumpMlPerSec =					212.0;
	EGMPrewashParam.MinPumpOnTime =					200;

/* Rinse*/
	EGMRinseParam.ReplenishingMode =							1;
	EGMRinseParam.ReplenishmentPerSqm =						500.0;
	EGMRinseParam.ReplenishmentPerPlate = 						150.0;
	EGMRinseParam.ReplenishmentIntervall = 						0;
	EGMRinseParam.PumpMlPerSec =								212.0;
	EGMRinseParam.MinPumpOnTime =							200;

/* Plate types*/
	for (i=0;i<MAXPLATETYPES;i++)
	{
		itoa(i,(UDINT )&tmpstr[0]);
		strcpy(EGMPlateTypes[i].Name,"Plate ");
		strcat(EGMPlateTypes[i].Name,tmpstr);
		strcpy(EGMPlateTypes[i].ManufacturerName,"Company");

		EGMPlateTypes[i].SizeX	= 					312.0;
		EGMPlateTypes[i].SizeY	= 					512.0;
		EGMPlateTypes[i].Area	= 					0.16;
		EGMPlateTypes[i].RegenerationPerSqrM	= 	0.0;
		EGMPlateTypes[i].RegenerationPerPlate	= 	0.0;
		EGMPlateTypes[i].Type	= 					i;
		EGMPlateTypes[i].DipTime	= 				0.0;
	}

	OverallPlateCounter =					0;
	OverallSqmCounter =					0;
	OverallReplenisherCounter =			0;
	ReplenisherCounter =					0;
	OverallReplenisherPumpTime =			0;
	DeveloperChangeDate =				OnTime;
	ReplenisherUsedSinceDevChange =		0;
	SqmSinceDevChg =						0;

	strcpy(MagicNumber,"Herbert");
}

_INIT void init(void)
{

Created = 0;
                        DInfo.enable      = 1;
                        DInfo.pDevice   = (UDINT) "ROOT";
                        DInfo.pPath     = (UDINT) "USER";

                        /* Call FUB */
                        DirInfo(&DInfo);

                        /* Get FUB output information */
                        wStatus         = DInfo.status;
                        dwDirNum        = DInfo.dirnum;
                        dwFileNum       = DInfo.filenum;
		if (wStatus ==fiERR_DIR_NOT_EXIST)
		{
			DCreate.enable = 1;
			DCreate.pDevice   = (UDINT) "ROOT";
			DCreate.pName = (UDINT) "USER";
			DirCreate(&DCreate);
			wStatus = DCreate.status;
			if (wStatus == 0)
				Created = 1;

		}

		DontResetMotorData = 0;
		PutTmpDataToSRAM = 0;
		GetTmpDataFromSRAM = 0;
	    saveParameterData = 0;
	    saveXData = 0;
	    saveMotorData = 0;
		savePlatesMade = 0;

	    put.enable=1;
	    get.enable=1;
	    loadParameterData = 1;
		loadPlatesMade = 1;
		loadMotorData = 1;
		StartUp = 1;
		ReadActive = 0;
		WriteActive=0;
		SaveToFile = 0;
		TmpPtr = &tmp[0];
/*V1.95 make sure, all numbers are correct*/
		for(i = 0; i < MAXTROLLEYS; i++)
		{
			Trolleys[i].Number 	= i;
		}
		for(i = 0; i < MAXPLATETYPES; i++)
		{
			PlateTypes[i].Number = i;
		}
}

_CYCLIC void zykl ()
{
	Test1 = sizeof(DeloaderParameter);
	Test2= sizeof (Motors);

	if(!loadMotorData && !loadParameterData && !loadXData && StartUp)
	{
		/*Machine number valid? (not "12345" AND defaults ok?*/
#ifdef MODE_BLUEFIN
	/*MagicNumber OK-> Daten im SRAM gültig-> Datei schreiben*/
		if( !strcmp(MagicNumber,"Herbert") )
#else
		if( memcmp(GlobalParameter.MachineNumber,"12345",5) && !strcmp(Motors[MAXMOTORS].Parameter.Function,"Krause-Biagosch") )
#endif
		{
		/*save sram to file*/
			SaveToFile = 1;
		}
		else
		{
		/*try to load sram from file*/
			FileIOData = (UDINT *) &tmp[0];
			FileIOLength = sizeof(tmp);
			strcpy(FileType,"SAV");
			strcpy(FileIOName,"SRAM");

			if(!ReadActive)
			{
				ReadActive = 1;
				ReadFileCmd = 1;
				ReadFileOK = 0;
				FileNotExisting = 0;
			}
			else
			{
/*wait for reading ready*/
				if(ReadFileOK)
				{
					ReadActive = 0;
					ReadFileOK = 0;
					StartUp = 0;
					/*save to SRAM*/
				    put.offset=0;
					put.len = OVERALLSRAMSIZEWORDS; /*WORDS!!*/
					put.address=(UDINT) &tmp[0];
					SRAMPut (&put);
					loadMotorData = 1;
					loadParameterData = 1;
					loadXData = 1;
					loadPlatesMade = 1;
				}
/*file not existing*/
				if(FileNotExisting)
				{
					Test1 = 123;
/*no defaults: set defaults*/
					if(strcmp(Motors[MAXMOTORS].Parameter.Function,"Krause-Biagosch") )
					{
						InitMotorData();
						InitXData();
						InitGlobalData();
						strcpy(Motors[MAXMOTORS].Parameter.Function,"Krause-Biagosch");
						saveMotorData = 1;
						saveParameterData = 1;
						saveXData = 1;
						savePlatesMade = 1;
					}
/*no file: set defaults*/
					EGMSetDefaults();
					ReadActive = 0;
					ReadFileOK = 0;
					FileNotExisting = 0;
					StartUp = 0;

				}
			}
		}
	}

	if (saveXData)
	{
	    put.offset=0;
	    put.len=((sizeof (X_Param))/2)+1;
	    put.address=(UDINT) &X_Param;
	    SRAMPut (&put);
		saveXData = 0;
		SaveToFile = 1;
	}

	if (saveMotorData)
	{
	    put.offset=300;
	    put.len=((sizeof (Motors))/2)+1;
	    put.address=(UDINT) &Motors[0];
	    SRAMPut (&put);
	    saveMotorData = 0;
		SaveToFile = 1;
	}

	if (saveParameterData)
	{
/* Laserleistungstabelle*/
	    put.offset=3800;
	    put.len=((sizeof (LaserPowerSettings))/2)+1;
	    put.address=(UDINT) &LaserPowerSettings[0];
	    SRAMPut (&put);

	    put.offset=4000;
	    put.len=((sizeof (FeederParameter))/2)+1;
	    put.address=(UDINT) &FeederParameter;
	    SRAMPut (&put);

	    put.offset=4200;
	    put.len=((sizeof (PaperRemoveParameter))/2)+1;
	    put.address=(UDINT) &PaperRemoveParameter;
	    SRAMPut (&put);

	    put.offset=4600;
	    put.len=((sizeof (AdjusterParameter))/2)+1;
	    put.address=(UDINT) &AdjusterParameter;
	    SRAMPut (&put);

	    put.offset=4800;
	    put.len=((sizeof (GlobalParameter))/2)+1;
	    put.address=(UDINT) &GlobalParameter;
	    SRAMPut (&put);

	    put.offset=5000;
	    put.len=((sizeof (PlateParameter))/2)+1;
	    put.address=(UDINT) &PlateParameter;
	    SRAMPut (&put);

	    put.offset=5200;
	    put.len=((sizeof (DeloaderParameter))/2)+1;
	    put.address=(UDINT) &DeloaderParameter;
	    SRAMPut (&put);

	    put.offset=5400;
	    put.len=((sizeof (Trolleys))/2)+1;
	    put.address=(UDINT) &Trolleys[0];
	    SRAMPut (&put);

/*sizeof(Trolleys) = 800 + 200 spare*/

	    put.offset=6400;
	    put.len=((sizeof (PlateTypes))/2)+1;
	    put.address=(UDINT) &PlateTypes[0];
	    SRAMPut (&put);
/*sizeof(PlateTypes) = 840 */

	    put.offset=8980;
	    put.len=((sizeof (gVERSION))/2)+1;
	    put.address=(UDINT) &gVERSION[0];
	    SRAMPut (&put);

/************************************************/
/****** EGM Daten **********/
/************************************************/
	    put.offset=10010;
	    put.len=((sizeof (EGMGlobalParam))/2)+1;
	    put.address= (UDINT)&EGMGlobalParam;
	    SRAMPut (&put);

	    put.offset=10600;
	    put.len=((sizeof (EGMAutoParam))/2)+1;
	    put.address=(UDINT)&EGMAutoParam;
	    SRAMPut (&put);

	    put.offset=10800;
	    put.len=((sizeof (EGMPreheatParam))/2)+1;
	    put.address=(UDINT) &EGMPreheatParam;
	    SRAMPut (&put);

	    put.offset=11000;
	    put.len=((sizeof (EGMDeveloperTankParam))/2)+1;
	    put.address=(UDINT) &EGMDeveloperTankParam;
	    SRAMPut (&put);

	    put.offset=11200;
	    put.len=((sizeof (EGMPlateTypes))/2)+1;
	    put.address=(UDINT) &EGMPlateTypes[0];
	    SRAMPut (&put);

	    put.offset=11700;
	    put.len=((sizeof (EGMPrewashParam))/2)+1;
	    put.address=(UDINT) &EGMPrewashParam;
	    SRAMPut (&put);

	    put.offset=11800;
	    put.len=((sizeof (EGMRinseParam))/2)+1;
	    put.address=(UDINT) &EGMRinseParam;
	    SRAMPut (&put);

	    put.offset=11890;
	    put.len=((sizeof (MagicNumber))/2)+1;
	    put.address=(UDINT) &MagicNumber[0];
	    SRAMPut (&put);

	    saveParameterData = 0;
		SaveToFile = 1;
	}

	if(savePlatesMade)
	{
/* 1.47
 * Nach jeder Belichtung werden jetzt auch die Trolleydaten gespeichert,
 * damit der Platten-Füllstand nach Aus- und Einschalten korrekt angezeigt wird
 */
	    put.offset=5400;
	    put.len=((sizeof (Trolleys))/2)+1;
	    put.address=(UDINT) &Trolleys[0];
	    SRAMPut (&put);

	    put.offset=9000;
	    put.len=(sizeof (UDINT))/2;
	    put.address=(UDINT) &PlatesMade;
	    SRAMPut (&put);
	    savePlatesMade = 0;
		SaveToFile = 1;
	}

	if( SaveToFile  )
	{
		/*save sram to file*/
		if(!WriteActive)
		{
			if ( !DeleteFileCmd && !ReadFileCmd && !WriteFileCmd && !WriteFileOK && (wBildNr != FILEPIC) && (wBildNr != MESSAGEPIC))
			{
				WriteActive = 1;
				get.offset=0;
				get.len = OVERALLSRAMSIZEWORDS; /*WORDS!!*/
				get.address=(UDINT) &tmp[0];
				SRAMGet (&get);

				FileIOData = (UDINT *) &tmp[0];
				FileIOLength = sizeof(tmp);
				strcpy(FileType,"SAV");
				strcpy(FileIOName,"SRAM");
				WriteFileCmd = 1;
				WriteFileOK = 0;
			}
			/*WriteFileCmd is true? just wait...*/
		}
		else
		{
		/*wait for writing ready*/
			if(WriteFileOK)
			{
				WriteActive = 0;
				SaveToFile = 0;
				StartUp = 0;
				WriteFileOK = 0;
				ParameterChanged = 1;
			}
		}
	}

/*******************************************************/
/* LOAD*/
/*******************************************************/

	if(loadXData)
	{
		len = sizeof (X_Param);
	    get.offset=0;
		get.len = (len / 2) +1;
		get.address=(UDINT) &tmp[0];
		SRAMGet (&get);
		memcpy(&X_Param,tmp,len);
	    loadXData = 0;
	}

	if(loadMotorData)
	{
		Motor_Typ BackupMotors[MAXMOTORS+1];
		len = sizeof (Motors);
		if (DontResetMotorData)
			memcpy(&BackupMotors[0],&Motors[0],len);

	    get.offset=300;
	    get.len=(len /2 ) +1;
	    get.address=(UDINT)&tmp[0];
	    SRAMGet (&get);
		memcpy(&Motors[0],tmp,len);
	    loadMotorData = 0;
	    if (DontResetMotorData)
	    {
			for (i = 0;i<=MAXMOTORS;i++)
			{
				Motors[i].Error = BackupMotors[i].Error;
				Motors[i].ReferenceOk = BackupMotors[i].ReferenceOk;
				Motors[i].Moving = BackupMotors[i].Moving;
				Motors[i].StartRef = BackupMotors[i].StartRef;
				Motors[i].ReferenceStep = BackupMotors[i].ReferenceStep;
				Motors[i].timeout = BackupMotors[i].timeout;
				Motors[i].Position = BackupMotors[i].Position;
				Motors[i].Position_mm = BackupMotors[i].Position_mm;
				Motors[i].LastPosition = BackupMotors[i].LastPosition;
			}
	    }
	    else
	    {
			for (i = 0;i<=MAXMOTORS;i++)
			{
				Motors[i].Error = 0;
				Motors[i].ReferenceOk = 0;
				Motors[i].Moving = 0;
				Motors[i].StartRef = 0;
				Motors[i].ReferenceStep = 0;
				Motors[i].timeout = 0;
				Motors[i].Position = 0;
				Motors[i].Position_mm = 0;
				Motors[i].LastPosition = 0;
			}
		}
		DontResetMotorData = 0;
	}

	if(loadParameterData)
	{
/* Laserleistungstabelle*/
		len = sizeof(LaserPowerSettings);
	    get.offset=3800;
	    get.len=(len / 2) +1;
	    get.address=(UDINT) &tmp[0];
	    SRAMGet (&get);
		memcpy(&LaserPowerSettings[0],tmp,len);

		len = sizeof(FeederParameter);
	    get.offset=4000;
	    get.len=(len / 2) +1;
	    get.address=(UDINT) &tmp[0];
	    SRAMGet (&get);
		memcpy(&FeederParameter,tmp,len);

		len = sizeof(PaperRemoveParameter);
	    get.offset=4200;
	    get.len=(len / 2) +1;
	    get.address=(UDINT) &tmp[0];
	    SRAMGet (&get);
		memcpy(&PaperRemoveParameter,tmp,len);
		 if (PaperRemoveParameter.PaperGripCycles>10)
		 	PaperRemoveParameter.PaperGripCycles = 2;

		len = sizeof(AdjusterParameter);
	    get.offset=4600;
	    get.len=(len / 2) +1;
	    get.address=(UDINT) &tmp[0];
	    SRAMGet (&get);
		memcpy(&AdjusterParameter,tmp,len);

		len = sizeof(GlobalParameter);
	    get.offset=4800;
	    get.len=(len / 2) +1;
	    get.address=(UDINT) &tmp[0];
	    SRAMGet (&get);
		memcpy(&GlobalParameter,tmp,len);
		Expose_Param.ScansPerMinute = GlobalParameter.ScansPerMinute;
		Expose_Param.Resolution  = GlobalParameter.Resolution;
		MirroredMachine = (GlobalParameter.MirroredMachine == 42);

/*safety bei update*/
		if ( (GlobalParameter.LaserPower != ((GlobalParameter.RealLaserPower+5) / 10))
			|| (GlobalParameter.RealLaserPower>1000)
		)
			GlobalParameter.RealLaserPower = GlobalParameter.LaserPower * 10;

		if( (GlobalParameter.DisableSlowMode != 0)
		 && (GlobalParameter.DisableSlowMode != 1) )
			GlobalParameter.DisableSlowMode = 1;

		if( GlobalParameter.SlowModeWaitTime > 9900 )
			GlobalParameter.SlowModeWaitTime = 2000;

		len = sizeof(PlateParameter);
	    get.offset=5000;
	    get.len=(len / 2) +1;
	    get.address=(UDINT) &tmp[0];
	    SRAMGet (&get);
		memcpy(&PlateParameter,tmp,len);
		if(isnan(PlateParameter.Length)) PlateParameter.Length = 0.0;
		if(isnan(PlateParameter.Width)) PlateParameter.Width = 0.0;
		if(isnan(PlateParameter.XOffset)) PlateParameter.XOffset = 0.0;
		if(isnan(PlateParameter.YOffset)) PlateParameter.YOffset = 0.0;
		if(isnan(PlateParameter.Thickness)) PlateParameter.Thickness = 0.0;
		if(isnan(PlateParameter.Sensitivity)) PlateParameter.Sensitivity = 0.0;
		len = sizeof(DeloaderParameter);
	    get.offset=5200;
	    get.len=(len / 2) +1;
	    get.address=(UDINT) &tmp[0];
	    SRAMGet (&get);
		memcpy(&DeloaderParameter,tmp,len);
		if( (DeloaderParameter.TableDeloadSpeed < 10.0) || (DeloaderParameter.TableDeloadSpeed > 1000.0) )
			DeloaderParameter.TableDeloadSpeed = 200.0;
		if( (DeloaderParameter.TableDeloadSpeedManual < 10.0) || (DeloaderParameter.TableDeloadSpeedManual > 1000.0) )
			DeloaderParameter.TableDeloadSpeedManual = 200.0;

		len = sizeof(Trolleys);
	    get.offset=5400;
	    get.len=(len / 2) +1;
	    get.address=(UDINT) &tmp[0];
	    SRAMGet (&get);
		memcpy(&Trolleys[0],tmp,len);
/*SAFETY*/
		for(i=0;i<MAXTROLLEYS;i++)
		{
			Trolleys[i].Name[MAXTROLLEYNAMELENGTH-1] = 0;
			Trolleys[i].Number 	= i;
			if(GlobalParameter.FlexibleFeeder == FALSE)
			{
				Trolleys[i].Double 	= 1;
				Trolleys[i].Single 	= 0;
				Trolleys[i].RightStack = 0;
			}

		}

		len = sizeof(PlateTypes);
	    get.offset=6400;
	    get.len=(len / 2) +1;
	    get.address=(UDINT) &tmp[0];
	    SRAMGet (&get);
		memcpy(&PlateTypes[0],tmp,len);
/*SAFETY*/
		for(i=0;i<MAXPLATETYPES;i++)
		{
			PlateTypes[i].Number = i;
			PlateTypes[i].Name[MAXPLATETYPENAMELENGTH-1] = 0;
			if(isnan(PlateTypes[i].Length)) PlateTypes[i].Length = 0.0;
			if(isnan(PlateTypes[i].Width)) PlateTypes[i].Width = 0.0;
			if(isnan(PlateTypes[i].XOffset)) PlateTypes[i].XOffset = 0.0;
			if(isnan(PlateTypes[i].YOffset)) PlateTypes[i].YOffset = 0.0;
			if(isnan(PlateTypes[i].Thickness)) PlateTypes[i].Thickness = 0.0;
			if(isnan(PlateTypes[i].Sensitivity)) PlateTypes[i].Sensitivity = 0.0;
			if (PlateTypes[i].SeparateBeltTracks > 1) PlateTypes[i].SeparateBeltTracks = 0;
		}

/************************************************/
/****** EGM Daten **********/
/************************************************/
	 	len = sizeof(EGMGlobalParam);
	    get.offset=10010;
	    get.len=(len / 2) +1;
	    get.address=(UDINT) &tmp[0];
	    SRAMGet (&get);
		memcpy(&EGMGlobalParam,tmp,len);
		strcpy(EGMGlobalParam.Version,gVERSION);
		if( (EGMGlobalParam.MachineType == BLUEFIN_XS)
		 || (EGMGlobalParam.MachineType == BLUEFIN_LOWCHEM) )
			MachineType = EGMGlobalParam.MachineType;
		else
			EGMGlobalParam.MachineType = MachineType;

	 	len = sizeof(EGMAutoParam);
	    get.offset=10600;
	    get.len=(len / 2) +1;
	    get.address=(UDINT) &tmp[0];
	    SRAMGet (&get);
		memcpy(&EGMAutoParam,tmp,len);

	 	len = sizeof(EGMPreheatParam);
	    get.offset=10800;
	    get.len=(len / 2) +1;
	    get.address=(UDINT) &tmp[0];
	    SRAMGet (&get);
		memcpy(&EGMPreheatParam,tmp,len);
		PreheatParamEnter = 1;

	 	len = sizeof(EGMDeveloperTankParam);
	    get.offset=11000;
	    get.len=(len / 2) +1;
	    get.address=(UDINT)&tmp[0];
	    SRAMGet (&get);
		memcpy(&EGMDeveloperTankParam,tmp,len);
		if(isnan(EGMDeveloperTankParam.PumpMlPerSec))
			EGMDeveloperTankParam.PumpMlPerSec = 20.0;
		if(isnan(EGMDeveloperTankParam.TopUpPumpMlPerSec))
			EGMDeveloperTankParam.TopUpPumpMlPerSec = 20.0;
		DeveloperTankParamEnter = 1;

	 	len = sizeof(EGMPlateTypes);
	    get.offset=11200;
	    get.len=(len / 2) +1;
	    get.address=(UDINT)&tmp[0];
	    SRAMGet (&get);
		memcpy(&EGMPlateTypes[0],tmp,len);

	 	len = sizeof(EGMPrewashParam);
	    get.offset=11700;
	    get.len=(len / 2) +1;
	    get.address=(UDINT)&tmp[0];
	    SRAMGet (&get);
		memcpy(&EGMPrewashParam,tmp,len);

	 	len = sizeof(EGMRinseParam);
	    get.offset=11800;
	    get.len=(len / 2) +1;
	    get.address=(UDINT)&tmp[0];
	    SRAMGet (&get);
		memcpy(&EGMRinseParam,tmp,len);

	 	len = sizeof(MagicNumber);
	    get.offset=11890;
	    get.len=(len / 2) +1;
	    get.address=(UDINT)&tmp[0];
	    SRAMGet (&get);
		memcpy(&MagicNumber[0],tmp,len);
/*
		if (strcmp(MagicNumber,"Herbert"))
			EGMSetDefaults();
*/

	    loadParameterData = 0;
	}

	if(loadPlatesMade)
	{
	    get.offset=9000;
	    get.len=(sizeof (UDINT))/2;
	    get.address=(UDINT) &PlatesMade;
	    SRAMGet (&get);
		loadPlatesMade = 0;
	}

	if(ClearSRAM)
	{
		for(i=0;i<OVERALLSRAMSIZEEBYTES;i++)
			tmp[i] = 255;
	    put.offset=0;
	    put.len=OVERALLSRAMSIZEWORDS;
	    put.address=(UDINT) &tmp[0];
	    SRAMPut (&put);
		ClearSRAM = 0;
	}

/* HA V1.50 give possibility to load SRAM from file */
/* to be used for copying data from one machine to another */
/*not used yet!*/
	if(LoadSRAMFromFile)
	{
		/*try to load sram from file*/
			FileIOData = (UDINT *) &tmp[0];
			FileIOLength = sizeof(tmp);
			strcpy(FileType,"SAV");
			strcpy(FileIOName,"SRAM");

			if(!ReadActive)
			{
				if ( !DeleteFileCmd && !ReadFileCmd && !WriteFileCmd && !ReadFileOK && (wBildNr != 42) && (wBildNr != MESSAGEPIC))
				{
					ReadActive = 1;
					ReadFileCmd = 1;
					ReadFileOK = 0;
					FileNotExisting = 0;
				}
			}
			else
			{
/*wait for reading ready*/
				if(ReadFileOK)
				{
					LoadSRAMFromFile = 0;
					ReadActive = 0;
					ReadFileOK = 0;
					/*save to SRAM*/
				    put.offset=0;
					put.len = OVERALLSRAMSIZEWORDS; /*WORDS!!*/
					put.address=(UDINT) &tmp[0];
					SRAMPut (&put);
					loadMotorData = 1;
					loadParameterData = 1;
					loadXData = 1;
					loadPlatesMade = 1;
				}

/*file not existing -> nothing happens*/
				if(FileNotExisting)
				{
					LoadSRAMFromFile = 0;
					ReadActive = 0;
					ReadFileOK = 0;
					FileNotExisting = 0;
				}
			}

	}

	if ( PutTmpDataToSRAM )
	{
		/*save to SRAM*/
	    put.offset=0;
		put.len = OVERALLSRAMSIZEWORDS; /*WORDS!!*/
		put.address=(UDINT) &tmp[0];
		SRAMPut (&put);
		loadMotorData = 1;
		DontResetMotorData = 1;
		loadParameterData = 1;
		loadXData = 1;
/*V2.00 gemachte Platten soll nicht mit geladen werden*/
/*		loadPlatesMade = 1;*/
		PutTmpDataToSRAM = 0;
		SaveToFile = 1;
	}

	if ( GetTmpDataFromSRAM )
	{
		get.offset=0;
		get.len = OVERALLSRAMSIZEWORDS; /*WORDS!!*/
		get.address=(UDINT) &tmp[0];
		SRAMGet (&get);
		GetTmpDataFromSRAM = 0;
	}

	if(GlobalParameter.Resolution != Expose_Param.Resolution)
	{
		GlobalParameter.Resolution = Expose_Param.Resolution;
		saveParameterData = 1;
	}
	if(GlobalParameter.ScansPerMinute != Expose_Param.ScansPerMinute)
	{
		GlobalParameter.ScansPerMinute = Expose_Param.ScansPerMinute;
		saveParameterData = 1;
	}

}
```

### Program Logical/ip_clt_c (ANSIC, version 1.00.0) - TCP IP Client

#### ip_clt_c.c
```c
#ifdef _DEFAULT_INCLUDES
	#include <AsDefault.h>
#endif
/****************************************************************************/
/*	TCP/IP Client Funktionalität 											*/
/*																			*/
/*																			*/
/*	Versionsgeschichte:														*/
/*  Version		Datum		Änderung								von		*/
/*	1.0			25.02.03	erste Implementation der				HA		*/
/*							Ping Funktion									*/
/*	1.10		26.02.03	SMTP Client								HA		*/
/*																			*/
/****************************************************************************/

/***** Include-Files: *****/
#include <bur/plc.h>
#include <bur/plctypes.h>
#include <string.h>
#include <Ethernet.h>
#include <EthSock.h>
#include "glob_var.h"
#include "asstring.h"

/***** Variablen-/Konstantendeklaration: *****/
/* Anwendungsspezifische Konstanten: */
#define SEND_BUFFER_LEN	128					/* Buffer-Länge für das Senden */
#define RECV_BUFFER_LEN	128					/* Empfangs-Buffer Länge */
#define SMTP_TIMEOUT	50

/* sonstige Konstanten */
#define TCP_IP_OK			0
#define TCP_IP_BUSY			65535

/*eigene Fehlermeldungen*/
#define	SERVER_CLOSED_CONN	1000
#define NO_CONNECTION		1001
#define SEND_TIMEOUT		1002

/*B+R Fehlermeldungen ethernet*/
#define ERR_ETH_INVAL 		27122
#define ERR_ETH_TIMEOUT		27160
#define ERR_ETH_CONNREFUSED	27161
#define ERR_ETH_NET_SLOW 	27210

/*B+R Fehlermeldungen ping*/
#define	PING_NO_RESPONSE	27220
#define	PING_TIMEOUT		27221

typedef struct
{
	STRING 	Server[16];
	STRING	Sender[60];
	STRING	Recipient[60];
	STRING	Subject[60];
	STRING	DataLine1[60];
	STRING	DataLine2[60];
	STRING	DataLine3[60];
	STRING	DataLine4[60];
	STRING	DataLine5[60];
	USINT	Step;
	USINT	CommStep;
	USINT	StartSending;
	UINT	TimeoutCounter;
	UINT	ErrorNr;
}SMTP_typ;

_LOCAL	SMTP_typ SMTP;

/* Strukturen fuer Ethernet-Libraray-Funktionen */
_LOCAL	TCPclient_typ		SMTP_Client;
_LOCAL	TCPrecv_typ			SMTP_Recv;
_LOCAL	TCPsend_typ			SMTP_Send;
_LOCAL	TCPclose_typ		SMTP_Close;

/* Variablen: */
_LOCAL	STRING	SendBuffer[SEND_BUFFER_LEN];
_LOCAL	STRING	RecvBuffer[RECV_BUFFER_LEN];

USINT PingOK,PingError;
_LOCAL	ICMPping_typ PingVar;
_LOCAL	UINT	PingOKInvisible,PingErrorInvisible;
_LOCAL USINT StartPing,IPAdr1,IPAdr2,IPAdr3,IPAdr4;
_LOCAL	UINT	MailAnimCounter;
UINT	AnimTimer,TryCounter;

STRING IPAdress[16],tmp[10];
TOF_10ms_typ PingLEDOff;
BOOL	Reconnect;

void Ping(void)
{
	PingOKInvisible = !PingOK;
	PingErrorInvisible = !PingError;
	PingLEDOff.IN = StartPing;
	PingLEDOff.PT = 300;
	TOF_10ms(&PingLEDOff);
	if(!PingLEDOff.Q)
	{
		PingOK = 0;
		PingError = 0;
	}
	if(StartPing)
	{
		PingVar.enable = TRUE;			/* FUB enable */
		strcpy(IPAdress,"");
		itoa(IPAdr1,(UDINT) &tmp[0]);
		strcat(IPAdress,tmp);
		strcat(IPAdress,".");
		itoa(IPAdr2,(UDINT) &tmp[0]);
		strcat(IPAdress,tmp);
		strcat(IPAdress,".");
		itoa(IPAdr3,(UDINT) &tmp[0]);
		strcat(IPAdress,tmp);
		strcat(IPAdress,".");
		itoa(IPAdr4,(UDINT) &tmp[0]);
		strcat(IPAdress,tmp);
		PingVar.ipaddr = inet_addr((UDINT)IPAdress);	/* IP Address of the Reciever */
		PingVar.timeout = 100;			/* Time of waiting */
		PingOK = 0;
		PingError = 0;
		ICMPping(&PingVar);
		switch(PingVar.status)
		{
			case 0:
			{
				/* Ping OK */
				StartPing = FALSE;
				PingOK = 1;
				PingError = 0;
				/***********************/
				/* TODO: Go on working */
				/***********************/
				break;
			}
			case TCP_IP_BUSY:
				/* Fub is already working */
				/* call again */
				break;
			case PING_NO_RESPONSE:
			{
				/* No Response */
				/*************************/
				/* TODO: Failure routine */
				/*************************/
				StartPing = FALSE;
				PingError = 1;
				PingOK = 0;
				break;
			}
			case PING_TIMEOUT:
			{
				/* Response timedout */
				/***************************/
				/* TODO: Failure routine   */
				/*		 Timeout to short? */
				/***************************/
				StartPing = FALSE;
				PingError = 1;
				PingOK = 0;
				break;
			}
			default:
			{
				/* Error occurs */
				StartPing = FALSE;
				/*************************/
				/* TODO: Failure routine */
				/*************************/
				PingError = 1;
				PingOK = 0;
				break;
			}
		}
	}
}

/***** INIT FUNKTION *******************************************************/
_INIT void init (void)
{
	strcpy(SMTP.Sender,"");
	strcpy(SMTP.Recipient,"");
	IPAdr1 = 192;
	IPAdr2 = 168;
	IPAdr3 = 77;
	IPAdr4 = 99;
} /* Ende Funktion _INIT void init (void) */

/***** ZYKLISCHE FUNKTION **************************************************/
_CYCLIC void cyclic (void)
{
	Ping();

/*V2.00 Mail-Funktion disabled (Bilder entfernt)*/
/*	Mail(); */

} /* Ende Funktion _CYCLIC void cyclic (void) */

/* ENDE */
```

### Program Logical/system (ANSIC, version 1.00.0) - System Einstellungen vornehmen

#### ip_chg.c
```c
#ifdef _DEFAULT_INCLUDES
	#include <AsDefault.h>
#endif
/****************************************************************************/
/*	IP Adresse und subnet mask setzen 										*/
/*	Achtung: Zum Einstellen des Gateway ist AR102 Version 2.61 erforderlich!*/
/*																			*/
/*	Versionsgeschichte:														*/
/*  Version		Datum		Änderung								von		*/
/*	1.0			28.02.03	erste Implementation 					HA		*/
/*																			*/
/****************************************************************************/

/***** Include-Files: *****/
#include <bur/plc.h>
#include <bur/plctypes.h>
#include "sys_lib.h"
#include "brsystem.h"
#include "AsArcfg.h"
#include <string.h>
#include "glob_var.h"
#include "asstring.h"
#include "Auxfunc.h"

#define NOERROR	0
#define cfgCONFIGMODE_MANUALLY 0
#define cfgERR_PARAM_NOT_SET 29009
#define cfgERR_SET_NOT_POSSIBLE 29004
#define ERR_FUB_BUSY 65535
#define ERR_VALUE_INVALID 29003

typedef struct
{
	char byte[4];
}IP_typ;

_LOCAL IP_typ	IPBytes;

_LOCAL UINT				SetIPStep;
_LOCAL	STRING		NewIP[16];
_LOCAL	USINT		SetIP,GetIP;

_LOCAL	STRING		OldIP[16],OldGateway[16],OldSubnet[16],entry[50],tmp[20];
_LOCAL	CfgGetIPAddr_typ CfgGetIPAddr_var;
_LOCAL	CfgSetIPAddr_typ CfgSetIPAddr_var;
_LOCAL	CfgGetDefaultGateway_typ CfgGetDefaultGateway_var;
_LOCAL	CfgSetDefaultGateway_typ CfgSetDefaultGateway_var;
_LOCAL	CfgGetSubnetMask_typ CfgGetSubnetMask_var;
_LOCAL	CfgSetSubnetMask_typ CfgSetSubnetMask_var;

_LOCAL CfgSetEthConfigMode_typ CfgSetEthConfigMode_var;

_LOCAL	USINT	IPAdr1,IPAdr2,IPAdr3,IPAdr4;
_LOCAL	USINT	Gateway1,Gateway2,Gateway3,Gateway4;
_LOCAL	USINT	Subnet1,Subnet2,Subnet3,Subnet4;
		BOOL	changed;

_LOCAL STRING OSVersionString[10];
_LOCAL TARGETInfo_typ TARGETInfo_01;
_LOCAL int ErrorCode;
int WaitCounter;
_GLOBAL USINT		gTriggerRedraw;

void IPString2Bytes(char *IPString,IP_typ *IP)
{
	int i,j,cnt;
	char help[16];
	i=0;
	j=0;
	cnt = 0;

	while(cnt<=3)
	{
		j=0;
		while( IPString[i]!='.' && IPString[i]!= 0 && i<16)
		{
			help[j] = IPString[i];
			i++;
			j++;
		/*safety!*/
			if(i>15) break;
		}
		help[j] = 0;
		IP->byte[cnt] = (char) atoi((UDINT) &help);
		cnt++;
		i++;
		if(i>15) break;
	}
}

void Bytes2IPString(char *IPStr,int Adr1,
								int Adr2,
								int Adr3,
								int Adr4)
{
	strcpy(IPStr,"");
	itoa(Adr1,(UDINT) &tmp[0]);
	strcat(IPStr,tmp);
	strcat(IPStr,".");
	itoa(Adr2,(UDINT) &tmp[0]);
	strcat(IPStr,tmp);
	strcat(IPStr,".");
	itoa(Adr3,(UDINT) &tmp[0]);
	strcat(IPStr,tmp);
	strcat(IPStr,".");
	itoa(Adr4,(UDINT) &tmp[0]);
	strcat(IPStr,tmp);
}

_INIT void init(void)
{
	GetIP = 0;
	SetIP = 0;
	SetIPStep = 0;
}

_CYCLIC void cyclic(void)
{
	if(xBildInit && (wBildAktuell == 124 || wBildAktuell == 11) )
		GetIP = 1;

	switch (SetIPStep)
	{
		case 0:
		{
			changed = 0;
	/*wait for start cmd*/
			if(GetIP)
			{
				SetIPStep = 5;
				strcpy(OldIP,"");
				strcpy(OldGateway,"");
				strcpy(OldSubnet,"");
				gTriggerRedraw = 1;
			}
			if(SetIP)
			{
				SetIPStep = 14;
			}
			break;
		}
/* aktuelle IP auslesen */
		case 5:
		{
			strcpy(entry,"IF5");
			CfgGetIPAddr_var.pDevice = (UDINT) &entry;
			CfgGetIPAddr_var.pIPAddr = (UDINT) &OldIP;
			CfgGetIPAddr_var.Len = 16;
			CfgGetIPAddr_var.enable = 1;
			CfgGetIPAddr(&CfgGetIPAddr_var);

			switch (CfgGetIPAddr_var.status)
			{
				case NOERROR:
				{
					IPString2Bytes(OldIP,&IPBytes);
					IPAdr1 = IPBytes.byte[0];
					IPAdr2 = IPBytes.byte[1];
					IPAdr3 = IPBytes.byte[2];
					IPAdr4 = IPBytes.byte[3];
					SetIPStep = 6;
					gTriggerRedraw = 1;
					break;
				}
				case ERR_FUB_BUSY:
					break;
			}
			break;
		}
/* aktuelles Def. Gateway auslesen */
		case 6:
		{
			strcpy(entry,"IF5");
			CfgGetDefaultGateway_var.pDevice = (UDINT) &entry;
			CfgGetDefaultGateway_var.pGateway = (UDINT) &OldGateway;
			CfgGetDefaultGateway_var.Len = 16;
			CfgGetDefaultGateway_var.enable = 1;
			CfgGetDefaultGateway(&CfgGetDefaultGateway_var);

			switch (CfgGetDefaultGateway_var.status)
			{
				case NOERROR:
				{
					IPString2Bytes(OldGateway,&IPBytes);
					Gateway1 = IPBytes.byte[0];
					Gateway2 = IPBytes.byte[1];
					Gateway3 = IPBytes.byte[2];
					Gateway4 = IPBytes.byte[3];
					SetIPStep = 7;
					gTriggerRedraw = 1;
					break;
				}
				case cfgERR_PARAM_NOT_SET:
				{
					SetIPStep = 7;
					break;
				}
				case ERR_FUB_BUSY:
					break;
				default:
				{
					ErrorCode = CfgGetDefaultGateway_var.status;
					break;
				}
			}
			break;
		}

/* aktuelles Def. Gateway auslesen */
		case 7:
		{
			strcpy(entry,"IF5");
			CfgGetSubnetMask_var.pDevice = (UDINT) &entry;
			CfgGetSubnetMask_var.pSubnetMask = (UDINT) &OldSubnet;
			CfgGetSubnetMask_var.Len = 16;
			CfgGetSubnetMask_var.enable = 1;
			CfgGetSubnetMask(&CfgGetSubnetMask_var);

			switch (CfgGetSubnetMask_var.status)
			{
				case NOERROR:
				{
					IPString2Bytes(OldSubnet,&IPBytes);
					Subnet1 = IPBytes.byte[0];
					Subnet2 = IPBytes.byte[1];
					Subnet3 = IPBytes.byte[2];
					Subnet4 = IPBytes.byte[3];
					SetIPStep = 13;
					gTriggerRedraw = 1;
					break;
				}
				case cfgERR_PARAM_NOT_SET:
				{
					SetIPStep = 13;
					break;
				}
				case ERR_FUB_BUSY:
					break;
				default:
				{
					ErrorCode = CfgGetSubnetMask_var.status;
					break;
				}
			}
			break;
		}

		case 13:
		{
			GetIP = 0;

		    TARGETInfo_01.enable = 1;                             /* Funktion wird nur ausgeführt wenn ENABLE <> 0
                                                             ist. */
		    TARGETInfo_01.pOSVersion = (UDINT) &OSVersionString;  /* Zeiger auf einen String mit vorgegebener Länge, in
                                                            den die Betriebssystemversion geschrieben wird */

		    TARGETInfo(&TARGETInfo_01);
			SetIPStep = 0;
			GetIP = 0;
			break;
		}

/******************************************************************/
/******************************************************************/
		case 14:
		{
			CfgSetEthConfigMode_var.enable = 1;
			CfgSetEthConfigMode_var.pDevice = (UDINT) &entry;
			CfgSetEthConfigMode_var.ConfigMode = cfgCONFIGMODE_MANUALLY;
			CfgSetEthConfigMode_var.Option = 1;
			CfgSetEthConfigMode(&CfgSetEthConfigMode_var);
			switch (CfgSetEthConfigMode_var.status)
			{
				case NOERROR:
				{
					SetIPStep = 15;
					break;
				}
				case ERR_FUB_BUSY:
					break;
				default:
				{
					ErrorCode = CfgSetEthConfigMode_var.status;
					break;
				}
			}
			break;
		}

/* set Subnetmask */
		case 15:
		{
			Bytes2IPString(NewIP,Subnet1,Subnet2,Subnet3,Subnet4);
			if( !strcmp(OldSubnet,NewIP) )
			{
				SetIPStep = 20;
				break;
			}

			strcpy(entry,"IF5");
			CfgSetSubnetMask_var.pDevice = (UDINT) &entry;
			CfgSetSubnetMask_var.pSubnetMask = (UDINT) &NewIP;
			CfgSetSubnetMask_var.Option = 1; /*NON-VOLATILE*/
			CfgSetSubnetMask_var.enable = 1;
			CfgSetSubnetMask(&CfgSetSubnetMask_var);

			switch (CfgSetSubnetMask_var.status)
			{
				case NOERROR:
				{
					SetIPStep = 20;
					break;
				}
				case cfgERR_SET_NOT_POSSIBLE:
				{
					SetIPStep = 20;
					break;
				}
				case ERR_FUB_BUSY:
					break;
				default:
				{
					ErrorCode = CfgSetSubnetMask_var.status;
					break;
				}
			}
			break;
		}

/* IP Adresse auf Änderung prüfen und ggf. setzen  */

/* set IP */
		case 20:
		{
			Bytes2IPString(NewIP,IPAdr1,IPAdr2,IPAdr3,IPAdr4);
			if( !strcmp(OldIP,NewIP) )
			{
				SetIPStep = 25;
				break;
			}

			strcpy(entry,"IF5");
			CfgSetIPAddr_var.pDevice = (UDINT) &entry;
			CfgSetIPAddr_var.pIPAddr = (UDINT) &NewIP;
			CfgSetIPAddr_var.Option = 1; /*NON-VOLATILE*/
			CfgSetIPAddr_var.enable = 1;
			CfgSetIPAddr(&CfgSetIPAddr_var);

			switch (CfgSetIPAddr_var.status)
			{
				case NOERROR:
				{
					SetIPStep = 25;
					break;
				}
				case ERR_FUB_BUSY:
					break;
				default:
				{
					ErrorCode = CfgSetIPAddr_var.status;
					break;
				}
			}
			break;
		}
/* set Gateway */
		case 25:
		{
			Bytes2IPString(NewIP,Gateway1,Gateway2,Gateway3,Gateway4);
			if( !strcmp(OldGateway,NewIP) )
			{
				SetIPStep = 0;
				SetIP = 0;
				GetIP = 1;
				break;
			}

			strcpy(entry,"IF5");
			CfgSetDefaultGateway_var.pDevice = (UDINT) &entry;
			CfgSetDefaultGateway_var.pGateway = (UDINT) &NewIP;
			CfgSetDefaultGateway_var.Option = 1; /*NON-VOLATILE*/
			CfgSetDefaultGateway_var.enable = 1;
			CfgSetDefaultGateway(&CfgSetDefaultGateway_var);

			switch (CfgSetDefaultGateway_var.status)
			{
				case NOERROR:
				{
					SetIPStep = 0;
					SetIP = 0;
					GetIP = 1;
					break;
				}
				case cfgERR_SET_NOT_POSSIBLE:
				{
					SetIPStep = 0;
					SetIP = 0;
					GetIP = 1;
					break;
				}
				case ERR_FUB_BUSY:
					break;
				default:
				{
					ErrorCode = CfgSetDefaultGateway_var.status;
					SetIPStep = 0;
					SetIP = 0;
					GetIP = 0;
					break;
				}
			}
			break;
		}

	}
}
```

### Program Logical/file (ANSIC, version 1.00.0) - File handling

#### file1.c
```c
#ifdef _DEFAULT_INCLUDES
	#include <AsDefault.h>
#endif
/****************************************************************************/
/*	Datei handling für Speichern/Laden von Einstellungen */
/*																			*/
/*																			*/
/*	Versionsgeschichte:														*/
/*  Version		Datum		Änderung								von		*/
/*	1.00		12.12.02	erste Implementation					HA		*/
/*	1.50		04.10.05	Statt Floppy jetzt Zugriff auf USB Stick*/
/*		*/
/*																			*/
/****************************************************************************/

/***** Header files *****/
#include <bur\plctypes.h>
#include <fileio.h>
#include <string.h>
#include "glob_var.h"
#include "auxfunc.h"

#define WEISS	4096
#define SCHWARZ	0

#define MAXFILES	50
#define MAXFILENAMELENGTH	32

#define READDIR		71
#define READDATA	73
#define WRITEDATA	72
#define NOFILE		74

/***** Variable declaration *****/
_LOCAL USINT byStep, byErrorLevel;
_LOCAL UDINT dwIdent;
_LOCAL UINT wStatus;
_LOCAL FileOpen_typ FOpen;
_LOCAL FileClose_typ FClose;
_LOCAL FileCreate_typ FCreate;
_LOCAL FileRead_typ FRead;
_LOCAL FileWrite_typ FWrite;
_LOCAL FileDelete_typ FDelete;

_GLOBAL	STRING FileIOName[MAXFILENAMELENGTH];
_GLOBAL	STRING	FileType[5];
_GLOBAL	UDINT *FileIOData;
_GLOBAL	UDINT	FileIOLength;
_GLOBAL	BOOL	WriteFileCmd,ReadFileCmd,DeleteFileCmd,WriteFileOK,ReadFileOK,DeleteFileOK,
				FileNotExisting,ReadDirCmd,ReadDirOK,NoDisk;

/***** Variable declaration *****/
_LOCAL UDINT 		dwDirNum, dwFileNum, dwCounter;
_LOCAL DirInfo_typ 	DInfo;
_LOCAL DirRead_typ 	DRead;
_LOCAL fiDIR_READ_DATA 	ReadData[MAXFILES];
_LOCAL	STRING	FileNames[MAXFILES][MAXFILENAMELENGTH];
_LOCAL	STRING Device[10];
_LOCAL BOOL	ReadDirData,ReadDirFloppy,DeleteFile,SelectionEnd;
_LOCAL	SINT	FileListPointer;
_LOCAL	UINT	DeviceDataInvisible,DeviceFloppyInvisible;

		BOOL	FirstTime,ReadDataActive,DeleteActive;
_LOCAL	UINT	DiskButtonPressed1,DiskButtonPressed2,FloppyButtonPressed1,FloppyButtonPressed2,
				DelButtonPressed1,DelButtonPressed2,FloppyInvisible,DeleteInvisible;
STRING	TmpFileName[MAXFILENAMELENGTH];
int FileListCounter;
BOOL	AbfrageAktiv;
_LOCAL UINT	HideWait,MessageNumber,Progress;
_LOCAL STRING FileNameDisplay[30];
_GLOBAL	UINT	DeviceType;
UINT	CycleCounter;

/***** Init part *****/
_INIT void Init(void)
{
	NoDisk = 0;
	/* Initialize variables */
	byStep 		= 0;
	byErrorLevel	= 0;

	/* Initialize file enable bits*/
	FOpen.enable 	= 1;
	FClose.enable 	= 1;
	FCreate.enable 	= 1;
	FRead.enable 	= 1;
	FWrite.enable 	= 1;
	FDelete.enable 	= 1;
	WriteFileOK = 0;
	ReadFileOK = 0;
	WriteFileCmd = 0;
	ReadFileCmd = 0;
	FileNotExisting = 0;
	ReadDirCmd = 0;
	ReadDirOK = 0;
	DeviceFloppyInvisible = 1;
	DeviceDataInvisible = 1;
	FirstTime = 1;
	DeleteFile = 0;
	DeleteActive = 0;
	strcpy(Device,"DATA");
	DelButtonPressed1 = WEISS;
	DelButtonPressed2 = SCHWARZ;
	DiskButtonPressed1 = WEISS;
	DiskButtonPressed2 = SCHWARZ;
	FloppyButtonPressed1 = WEISS;
	FloppyButtonPressed2 = SCHWARZ;
	HideWait = 1;
}

/***** Cyclic part *****/
_CYCLIC void Cyclic(void)
{
	if (!strcmp(Device,"DATA"))
		DeviceType = 0; /* CF Card*/
	else
		DeviceType = 1; /* USB */

	if(UserLevel < 2)
	{
		DeleteInvisible = 1;
		DeleteFile = 0;
	}
	else
	{
		FloppyInvisible = 0;
		DeleteInvisible = 0;
	}

	if(FileListPointer >= FileListCounter )FileListPointer = FileListCounter-1;
	if(SelectionEnd)
	{
		if(FileListPointer < 0)
			FileListPointer = FileListCounter-1;

		if(FileListPointer >= FileListCounter || FileListPointer < 0)
			FileListPointer = 0;

		strcpy(FileIOName,FileNames[FileListPointer]);
		SelectionEnd = 0;
	}

	if(DeleteFile && !DeleteInvisible)
	{
		DelButtonPressed1 = SCHWARZ;
		DelButtonPressed2 = WEISS;

		if( !AbfrageAktiv)
		{
			ShowMessage(101,1,0,REQUEST,OKCANCEL, FALSE);
/*
			if(wBildAktuell != MESSAGEPIC )
				OrgBild = wBildAktuell;
			wBildNeu = MESSAGEPIC;
			AbfrageOK = 0;
			AbfrageCancel = 0;
			IgnoreButtons = 0;
			OK_CancelButtonInv = 0;
			OK_ButtonInv = 1;
			AbfrageText1 = 102;
			AbfrageText2 = 1;
			AbfrageText3 = 0;
			AbfrageIcon = REQUEST;*/
			AbfrageAktiv = 1;
		}
		else
		{
			if(AbfrageOK)
			{
				AbfrageOK = 0;
				DeleteActive = 1;
				DeleteFile = 0;
				strcpy(FileIOName,FileNames[FileListPointer]);
				if(strlen(FileIOName) > 0 && strlen(FileIOName) < MAXFILENAMELENGTH)
					DeleteFileCmd = 1;
				else
				{
					DeleteFile = 0;
					DelButtonPressed1 = WEISS;
					DelButtonPressed2 = SCHWARZ;
				}
				AbfrageAktiv = 0;
			}
			if(AbfrageCancel)
			{
				AbfrageCancel = 0;
				DeleteFile = 0;
				DelButtonPressed1 = WEISS;
				DelButtonPressed2 = SCHWARZ;
				AbfrageAktiv = 0;
			}

		}

	}

	if( DeleteActive == 1 )
	{
		if(DeleteFileOK)
		{
			DeleteFileOK = 0;
			DeleteActive = 0;
			ReadDirCmd = 1;
			ReadDirOK = 0;
			DelButtonPressed1 = WEISS;
			DelButtonPressed2 = SCHWARZ;
			FileListPointer = 0;
			strcpy(FileIOName,FileNames[FileListPointer]);
		}
	}

	if(FirstTime && wBildNr == FILEPIC)
	{
		DeleteFile = 0;
		DeleteActive = 0;
		ReadDirData = 1;
		FirstTime = 0;
		FileListPointer = 0;
		strcpy(FileIOName,FileNames[FileListPointer]);
		DelButtonPressed1 = WEISS;
		DelButtonPressed2 = SCHWARZ;
	}
	if(wBildAktuell != FILEPIC && wBildAktuell != MESSAGEPIC)
		FirstTime = 1;

	if((ReadDirData || (ReadDirFloppy && !FloppyInvisible)) && !ReadDataActive)
	{
		ReadDirCmd = 1;
		ReadDirOK = 0;
		ReadDataActive = 1;
	}

	if(ReadDataActive)
	{
		if( ReadDirOK )
		{
			ReadDirOK = 0;
			ReadDataActive = 0;
			DiskButtonPressed1 = WEISS;
			DiskButtonPressed2 = SCHWARZ;
			FloppyButtonPressed1 = WEISS;
			FloppyButtonPressed2 = SCHWARZ;
			FileListPointer = 0;
			strcpy(FileIOName,FileNames[FileListPointer]);
		}
		if(NoDisk)
		{
			ReadDataActive = 0;
			ReadDirData = 1;
			strcpy(FileNames[0],"NO DISK!");
			NoDisk = 0;
			FileListPointer = 0;
			DiskButtonPressed1 = WEISS;
			DiskButtonPressed2 = SCHWARZ;
			FloppyButtonPressed1 = WEISS;
			FloppyButtonPressed2 = SCHWARZ;
		}
	}

	switch (byStep)
	{

		case 0:
		{

			if(!WriteFileCmd && !ReadFileCmd &&  !DeleteFileCmd && !ReadDirCmd)
			{
				HideWait = 1;
				break;
			}
/*safety: if both commands: read is preferred*/
			if(WriteFileCmd && ReadFileCmd)
				WriteFileCmd = 0;
			if( DeleteFileCmd )
			{
				byStep = 40;
				break;
			}
			if(ReadDirCmd)
			{
				byStep = 100;
				ReadDirOK = 0;
				HideWait = 0;
				MessageNumber = READDIR;
				break;
			}

			FileNotExisting = 0;
			WriteFileOK = 0;
			ReadFileOK = 0;
			DeleteFileOK = 0;
/*wenn SRAM Daten automatisch gespeichert werden, dann immer auf CF !*/
			if (!strcmp(FileType,"SAV"))
				strcpy(Device,"DATA");
	/* Initialize file open structrue */
			FOpen.pDevice 	= (UDINT) Device;

			strcpy(TmpFileName,FileIOName);
			strcat(TmpFileName,".");
			strcat(TmpFileName,FileType);
			FOpen.pFile 	= (UDINT) &TmpFileName[0]; 	/* File name */
			FOpen.mode 	= FILE_RW; 		/* Read and write access */
			/* Call FUB */
			FileOpen(&FOpen);

			/* Get FUB output information */
			dwIdent = FOpen.ident;
			wStatus = FOpen.status;

			if (wStatus == 65535)
			{
		/*wait */
				break;
			}

			if (wStatus == fiERR_FILE_NOT_FOUND )
			{
				if(ReadFileCmd)
				{
					ReadFileCmd = 0;
					FileNotExisting = 1;
					break;
				}
				if(!WriteFileCmd)
				{
					break;
				}
				else
				{
/*File does not exist->create it*/
					byStep = 5;
					HideWait = 0;
					MessageNumber = WRITEDATA;
					break;
				}
			}
			else if (wStatus != 0)
			{
				byStep = 50;
				WriteFileCmd = 0;
			}

/* no error, go ahead*/
			if( WriteFileCmd )
			{
				byStep = 10;
				HideWait = 0;
				MessageNumber = WRITEDATA;
			}
			if( ReadFileCmd )
			{
				byStep = 20;
				HideWait = 0;
				MessageNumber = READDATA;
			}

			FClose.ident 	= dwIdent;
			FRead.ident 	= dwIdent;
			FWrite.ident 	= dwIdent;

			break;
		}

		case 5: /**** create file ****/
		{
			/* Initialize file create structure */
			FCreate.enable 	= 1;
			FCreate.pDevice = (UDINT) Device;
			strcpy(TmpFileName,FileIOName);
			strcat(TmpFileName,".");
			strcat(TmpFileName,FileType);
			FCreate.pFile 	= (UDINT) &TmpFileName[0]; 	/* File name */

		/* Call FUB */
			FileCreate(&FCreate);

		/* Get output information of FUB */
			dwIdent = FCreate.ident;
			wStatus = FCreate.status;

			if (wStatus == 65535)
			{
		/*wait */
				break;
			}

			/* any error-> error message */
			if (wStatus != 0)
			{
				byStep = 50;
				WriteFileCmd = 0;
				break;
			}

			FClose.ident 	= dwIdent;
			FRead.ident 	= dwIdent;
			FWrite.ident 	= dwIdent;
			byStep = 10;
			break;
		}

		case 10: /**** Write data to file ****/
		{
			/* Initialize file write structure */
			FWrite.offset 	= 0;
			FWrite.pSrc 	= (UDINT) FileIOData;
			FWrite.len 	= FileIOLength;

			/* Call FUB */
			FileWrite(&FWrite);

			/* Get status */
			wStatus = FWrite.status;

			if (wStatus == 65535)
			{
				break;
			}

			/* any error -> error message */
			if (wStatus != 0)
			{
				byStep 		= 50;
				WriteFileCmd = 0;
			}
			else
			{
				byStep = 30; 	/* Set new step value : close*/
			}

			break;
		}

		case 20: /**** Read data from file ****/
		{
			/* Initialize file read structure */
			FRead.offset 	= 0;
			FRead.pDest 	= (UDINT) FileIOData;
			FRead.len 	= FileIOLength;

			/* Call FUB */
			FileRead(&FRead);

			/* Get status */
			wStatus = FRead.status;

			if (wStatus == 65535)
			{
				break;
			}

			/* any error -> error message*/
			if (wStatus != 0)
			{
				byStep = 50;
			}
			else
			{
				byStep = 30; 	/* Set new step value : close*/
			}

			break;
		}

		case 30: /**** Close file ****/
		{
			/* Initialize file close structure */
			FClose.ident 	= dwIdent;

			/* Call FUB */
			FileClose(&FClose);

			/* Get status */
			wStatus = FClose.status;

			if (wStatus == 65535)
			{
				break;
			}

			/* any error -> error message */
			if (wStatus != 0)
			{
				byStep = 50;
			}
			else
			{
				byStep = 0;	/* Set new step value */
				HideWait = 1;
				if(WriteFileCmd)
				{
					WriteFileCmd = 0;
					WriteFileOK = 1;
				}
				if(ReadFileCmd)
				{
					ReadFileCmd = 0;
					ReadFileOK = 1;
				}
			}

			break;
		}

		case 40: /**** Delete file ****/
		{
			/* Initialize file delete structure */
			FDelete.pDevice = (UDINT) Device;
			strcpy(TmpFileName,FileIOName);
			strcat(TmpFileName,".");
			strcat(TmpFileName,FileType);
			FDelete.pName 	= (UDINT) &TmpFileName[0]; 	/* File name */

			/* Call FUB */
			FileDelete(&FDelete);

			/* Get status */
			wStatus = FDelete.status;

			/* Verify status */
			if (wStatus == 65535)
			{
				break;
			}

			/* Verify status */
			if (wStatus == 26205)
			{
				FileNotExisting = 1;
			}
			else
			if(wStatus != 0)
				byErrorLevel = 6; 	/* Set error level for FileDelete */
			else
			{
				DeleteFileOK = 1;
			}
			byStep = 0; 						/* Reset step variable */
			DeleteFileCmd = 0;
			break;
		}

		case 50: /* ERROR */
		{
			HideWait = 1;
			ShowMessage(0,70,0,CAUTION,OKONLY, FALSE);
/*
			if(wBildAktuell != MESSAGEPIC )
				OrgBild = wBildAktuell;
			wBildNeu = MESSAGEPIC;
			AbfrageOK = 0;
			AbfrageCancel = 0;
			IgnoreButtons = 0;
			OK_CancelButtonInv = 1;
			OK_ButtonInv = 0;
			AbfrageText1 = 0;
			AbfrageText2 = 70;
			AbfrageText3 = 0;
			AbfrageIcon = CAUTION;*/
			byStep = 51;
			break;
		}
		case 51: /* wait for user reaction*/
		{
			if(AbfrageOK || AbfrageCancel)
				byStep = 0;

			break;
		}

/*********************************************/
/*Directory information*/
/*********************************************/
		case 100: /* read DIR Info */
		{
			int i;

			for(i=0;i<MAXFILES;i++)
				FileNames[i][0] = 0;
			if(ReadDirData)
			{
				strcpy(Device,"DATA");
				DeviceFloppyInvisible = 1;
				DeviceDataInvisible = 0;
				DiskButtonPressed1 = SCHWARZ;
				DiskButtonPressed2 = WEISS;
			}
			if(ReadDirFloppy && !FloppyInvisible)
			{
				strcpy(Device,"USBStick");
				DeviceFloppyInvisible = 0;
				DeviceDataInvisible = 1;
				FloppyButtonPressed1 = SCHWARZ;
				FloppyButtonPressed2 = WEISS;
			}

	/* Initialize info structure */
			DInfo.enable 	= 1;
			DInfo.pDevice 	= (UDINT) Device;
			DInfo.pPath 	= 0;

	/* Call FUB */
			DirInfo(&DInfo);

	/* Get FUB output information */
			wStatus 	= DInfo.status;
			dwDirNum 	= DInfo.dirnum;
			dwFileNum 	= DInfo.filenum;

			if (wStatus == 65535)
			{
				/*busy: just wait*/
				break;
			}

	/* Verify status */
			if (wStatus == fiERR_FILE_DEVICE)
			{
/* V4.02 if 1st USB device fails, check 2nd*/
				if (ReadDirFloppy)
				{
					byStep = 102;
				}
				else
				{
					NoDisk = 1;
					ReadDirCmd = 0;
					ReadDirOK = 0;
					byStep = 0;
					ReadDirFloppy = 0;
					ReadDirData = 0;
					HideWait = 1;
				}
			}
			else
			if (wStatus != 0)
			{
				ReadDirCmd = 0;
				ReadDirOK = 0;
				ReadDirFloppy = 0;
				ReadDirData = 0;
				HideWait = 1;
				byStep = 50;
			}
			else
			{
				NoDisk = 0;

	/* Verify number of found files */
				if (dwFileNum > MAXFILES)
				{
					dwFileNum = MAXFILES; 	/* Set variable to maximum value */
				}
				byStep = 105;
				dwCounter = 0;
				FileListCounter = 0;
			}
			break;
		}

		case 102: /* read DIR Info 2nd USB Port*/
		{
			strcpy(Device,"USBStick2");

	/* Initialize info structure */
			DInfo.enable 	= 1;
			DInfo.pDevice 	= (UDINT) Device;
			DInfo.pPath 	= 0;

	/* Call FUB */
			DirInfo(&DInfo);

	/* Get FUB output information */
			wStatus 	= DInfo.status;
			dwDirNum 	= DInfo.dirnum;
			dwFileNum 	= DInfo.filenum;

			if (wStatus == 65535)
			{
				/*busy: just wait*/
				break;
			}

	/* Verify status */
			if (wStatus == fiERR_FILE_DEVICE)
			{
				HideWait = 1;
				NoDisk = 1;
				ReadDirCmd = 0;
				ReadDirOK = 0;
				byStep = 0;
				ReadDirFloppy = 0;
				ReadDirData = 0;

				ShowMessage(0,69,0,CAUTION,OKONLY, TRUE);

/*				if(wBildAktuell != MESSAGEPIC )
					OrgBild = wBildAktuell;
				wBildNeu = MESSAGEPIC;
				AbfrageOK = 0;
				AbfrageCancel = 0;
				IgnoreButtons = 1;
				OK_CancelButtonInv = 1;
				OK_ButtonInv = 0;
				AbfrageText1 = 0;
				AbfrageText2 = 69;
				AbfrageText3 = 0;
				AbfrageIcon = CAUTION;*/

			}
			else
			if (wStatus != 0)
			{
				HideWait = 1;
				ReadDirCmd = 0;
				ReadDirOK = 0;
				ReadDirFloppy = 0;
				ReadDirData = 0;
				byStep = 50;
			}
			else
			{
				NoDisk = 0;

	/* Verify number of found files */
				if (dwFileNum > MAXFILES)
				{
					dwFileNum = MAXFILES; 	/* Set variable to maximum value */
				}
				byStep = 105;
				dwCounter = 0;
				FileListCounter = 0;
			}
			break;
		}

		case 105: /* read DIR Info */
		{
			ReadDirFloppy = 0;
			ReadDirData = 0;

		/* Verify counter variable */
			while (dwCounter < dwFileNum)
			{
			/* Initialize read directory structure */
				DRead.enable 	= 1;
				DRead.pDevice 	= (UDINT) Device;
				DRead.pPath 	= 0;
				DRead.entry 	= dwCounter;
				DRead.option 	= FILE_FILE;
				DRead.pData 	= (UDINT) &ReadData[dwCounter];
				DRead.data_len 	= sizeof (ReadData[0]);

			/* Call FUB */
				DirRead(&DRead);

			/* Get status */
				wStatus = DRead.status;

				if (wStatus == 65535)
				{
					/*busy: just wait*/
					break;
				}

			/* Verify status */
				if (wStatus != 0)
				{
					ReadDirCmd = 0;
					ReadDirOK = 0;
					HideWait = 1;
					byStep = 50;
					break;
				}
				else
				{
					int i = strlen(ReadData[dwCounter].Filename);
					STRING TypeFound[5];
					USINT *p;

/* für info display */
					if (i<=28)
						strcpy(FileNameDisplay,ReadData[dwCounter].Filename);
					else
					{
						strncpy(FileNameDisplay,ReadData[dwCounter].Filename,25);
						FileNameDisplay[25]=0;
						strcat(FileNameDisplay,"...");
					}

					strcpy(TmpFileName,ReadData[dwCounter].Filename);

					while(i-->1)
					{
						if( TmpFileName[i] == '.' )
						{
							TmpFileName[i] = 0;
							p = &TmpFileName[i+1];
								strcpy(TypeFound,p);
							if( !strcmp(TypeFound,FileType) )
								strcpy(FileNames[FileListCounter++],TmpFileName);
							i=0;
						}
					}
					dwCounter ++;	/* Increase counter variable */
					Progress = (dwCounter*100)/dwFileNum;
				}
			}

			if (wStatus == 65535)
			{
				/*busy: just wait*/
				break;
			}
/* keine Datei gefunden*/
			if (!FileListCounter)
			{
				MessageNumber = NOFILE; /* no file found */
				byStep = 106;
				CycleCounter = 0;
			}
			else
			{
				byStep = 0;
				HideWait = 1;
			}
			ReadDirCmd = 0;
			ReadDirOK = 1;
			Progress = 0;
			strcpy(FileNameDisplay,"");
			break;
		}
		case 106: /* wait, to let user read the message*/
		{
			CycleCounter++;
			if(CycleCounter >= 15)	/* 3 sec */
			{
				CycleCounter = 0;
				byStep = 0;
				HideWait = 1;
			}
			break;
		}
	}
}
```

- auxfunc.h (reference to Logical/GlobalIncludes/auxfunc.h)

#### usb.c - not listed in the package file held
```c
/********************************************************************
 * COPYRIGHT --
 ********************************************************************
 * Programm: File
 * Datei: usb.c
 * Autor: Aden
 * Erstellt: 10. Dezember 2014
 *******************************************************************/

#include <bur/plctypes.h>
#ifdef _DEFAULT_INCLUDES
	#include <AsDefault.h>
#endif

#define _REPLACE_CONST
#include <asusb.h>
#include <fileio.h>
#include <string.h>
#include <AsBrStr.h>
#include "auxfunc.h"

/* //////////////////////////////////////////////////////////////////
// DEFINES
////////////////////////////////////////////////////////////////// */
#define TRUE 1
#define FALSE 0
#define MAXUSBDEVICES 32
#define SANDISK_VENDOR_ID 0x0781
#define SANDISK_PRODUCT_ID 0x7105
#define SANDISK_BCD 0x1033
#define USB_GETNODELIST 1
#define USB_SEARCHDEVICE 2
#define USB_DEVICELINK 3
#define USB_DEVICEUNLINK 4
#define USB_FILEACCESS 5
#define MSDEVICE "USBStick0"
#define PARAMDEVICE "/DEVICE="
#define MAXLOGMESSAGELENGTH (250)
/* //////////////////////////////////////////////////////////////////
// DECLARATION
////////////////////////////////////////////////////////////////// */
_LOCAL UsbNodeListGet_typ UsbNodeListGetFub;
_LOCAL UsbNodeGet_typ UsbNodeGetFub;
_LOCAL usbNode_typ usbDevice;
_LOCAL DevLink_typ DevLinkFub;
_LOCAL DevUnlink_typ DevUnlinkFub;
_LOCAL BOOL deviceLinked;
_LOCAL UDINT usbAttachDetachCount;
_LOCAL UINT usbAction,usbNodeIx;
_LOCAL UDINT usbNodeList[MAXUSBDEVICES];
_LOCAL UDINT usbNodeId;
//_LOCAL char szDevParamName[asusb_DEVICENAMELENGTH+sizeof(PARAMDEVICE)];
_LOCAL char szDevParamName[150];
extern _LOCAL UINT FloppyInvisible;
extern _LOCAL char USBDeviceStr[32];

static    char                tmpMsg[MAXLOGMESSAGELENGTH+1];
static    char                lclposstr[30];
static    UINT                USBDevCnt;

void LogMessage(char *ptr)
{
	return;
}
/* //////////////////////////////////////////////////////////////////
// INIT UP
////////////////////////////////////////////////////////////////// */
void usbinit(void)
{
	usbAttachDetachCount = 0;
	usbNodeIx = 0;
	usbAction = USB_GETNODELIST;
	strcpy(USBDeviceStr,MSDEVICE);
	USBDevCnt = 0;
}
/* //////////////////////////////////////////////////////////////////
// CYCLIC TASK
////////////////////////////////////////////////////////////////// */
void usbcyclic(void)
{
	switch (usbAction)
	{
		case USB_GETNODELIST:
			FloppyInvisible = TRUE;
			UsbNodeListGetFub.enable = 1;
			UsbNodeListGetFub.pBuffer = (UDINT)&usbNodeList;
			UsbNodeListGetFub.bufferSize = sizeof(usbNodeList);
			UsbNodeListGetFub.filterInterfaceClass = asusb_CLASS_MASS_STORAGE;
			UsbNodeListGetFub.filterInterfaceSubClass = asusb_SUBCLASS_SCSI_COMMAND_SET;

			UsbNodeListGet(&UsbNodeListGetFub);
			if (UsbNodeListGetFub.status != ERR_FUB_BUSY)
				usbAttachDetachCount = UsbNodeListGetFub.attachDetachCount;

			if (UsbNodeListGetFub.status == ERR_OK /*&& UsbNodeListGetFub.listNodes*/)
			{
				/* USB Device Attach or detach */
				usbAction = USB_SEARCHDEVICE;
				usbNodeIx = 0;
			}
			else
			if (UsbNodeListGetFub.status == asusbERR_BUFSIZE
				|| UsbNodeListGetFub.status == asusbERR_NULLPOINTER)
			{
				/* Error Handling */
				strcpy(tmpMsg,"FILE: Error during UsbNodeListGet: ");
				brsitoa(UsbNodeListGetFub.status,(UDINT)lclposstr);
				strcat(tmpMsg,lclposstr);
				LogMessage(tmpMsg);
			}
			break;
		case USB_SEARCHDEVICE:
			UsbNodeGetFub.enable = 1;
			UsbNodeGetFub.nodeId = usbNodeList[usbNodeIx];
			UsbNodeGetFub.pBuffer = (UDINT)&usbDevice;
			UsbNodeGetFub.bufferSize = sizeof(usbDevice);
			UsbNodeGet(&UsbNodeGetFub);
			if (UsbNodeGetFub.status == ERR_OK )
			{
				/* MASS_STORAGE on 1st ? */
				if ((strcmp (usbDevice.ifName, "/bd0") == 0))
				{
					/* Mass Storage on Port IF5 found */
					strcpy(szDevParamName,PARAMDEVICE);
					strcat (szDevParamName,usbDevice.ifName);
					usbNodeId = usbNodeList[usbNodeIx];
					usbAction = USB_DEVICELINK;
					LogMessage("FILE: USB device detected ");

					strcpy(tmpMsg,"Class= ");
					brsitoa(usbDevice.interfaceClass,(UDINT)lclposstr);
					strcat(tmpMsg,lclposstr);
					strcat(tmpMsg,", Subclass= ");
					brsitoa(usbDevice.interfaceSubClass,(UDINT)lclposstr);
					strcat(tmpMsg,lclposstr);
					strcat(tmpMsg,", Protocol= ");
					brsitoa(usbDevice.interfaceProtocol,(UDINT)lclposstr);
					strcat(tmpMsg,lclposstr);
					strcat(tmpMsg,", VendorID= ");
					brsitoa(usbDevice.vendorId,(UDINT)lclposstr);
					strcat(tmpMsg,lclposstr);
					strcat(tmpMsg,", ProductID= ");
					brsitoa(usbDevice.productId,(UDINT)lclposstr);
					strcat(tmpMsg,lclposstr);
					strcat(tmpMsg,", ReleaseVersion= ");
					brsitoa(usbDevice.bcdDevice,(UDINT)lclposstr);
					strcat(tmpMsg,lclposstr);
					strcat(tmpMsg,", if-name= ");
					strcat(tmpMsg,usbDevice.ifName);
					LogMessage(tmpMsg);

				}
				else
				{
					usbNodeIx++;
					if (usbNodeIx >= UsbNodeListGetFub.allNodes)
					{
						/* USB Device not found */
						usbAction = USB_GETNODELIST;
					}
				}
			}
			else if (UsbNodeGetFub.status == asusbERR_USB_NOTFOUND)
			{
				/* USB Device not found */
				usbAction = USB_GETNODELIST;
			}
			else if (UsbNodeGetFub.status == asusbERR_BUFSIZE
				|| UsbNodeGetFub.status == asusbERR_NULLPOINTER)
			{
				/* Error Handling */
				strcpy(tmpMsg,"FILE: Error during UsbNodeGet: ");
				brsitoa(UsbNodeGetFub.status,(UDINT)lclposstr);
				strcat(tmpMsg,lclposstr);
				LogMessage(tmpMsg);

			}
			break;
		case USB_DEVICELINK:
			DevLinkFub.enable = 1;
			DevLinkFub.pDevice = (UDINT)USBDeviceStr;
			DevLinkFub.pParam = (UDINT)szDevParamName;
			DevLink(&DevLinkFub);
			if (DevLinkFub.status == ERR_OK)
			{
				LogMessage("FILE: USB device linked ");
				usbAction = USB_FILEACCESS;
				deviceLinked = TRUE;
			}
			else
			if (DevLinkFub.status == fiERR_DEVICE_ALREADY_EXIST)
			{
				USBDevCnt++;
				if(USBDevCnt > 9)
					USBDevCnt = 0;
				USBDeviceStr[strlen(USBDeviceStr)-1] = USBDevCnt + '0';
			}
			else
			if (DevLinkFub.status != ERR_FUB_BUSY)
			{
				strcpy(tmpMsg,"FILE: Error during DevLink: ");
				brsitoa(DevLinkFub.status,(UDINT)lclposstr);
				strcat(tmpMsg,lclposstr);
				LogMessage(tmpMsg);
			}
			break;
		case USB_DEVICEUNLINK:
			DevUnlinkFub.enable = 1;
			DevUnlinkFub.handle = DevLinkFub.handle;
			DevUnlink(&DevUnlinkFub);
			if (DevUnlinkFub.status == ERR_OK)
			{
				LogMessage("FILE: USB device un-linked ");
				usbAction = USB_GETNODELIST;
				deviceLinked = FALSE;
			}
			else
			if (DevUnlinkFub.status != ERR_FUB_BUSY)
			{
				strcpy(tmpMsg,"FILE: Error during DevUnLink: ");
				brsitoa(DevUnlinkFub.status,(UDINT)lclposstr);
				strcat(tmpMsg,lclposstr);
				LogMessage(tmpMsg);
			}
			break;
		case USB_FILEACCESS:
			/* Check USB Device */
			UsbNodeGetFub.enable = 1;
			UsbNodeGetFub.nodeId = usbNodeId;
			UsbNodeGetFub.pBuffer = (UDINT)&usbDevice;
			UsbNodeGetFub.bufferSize = sizeof(usbDevice);
			UsbNodeGet(&UsbNodeGetFub);
			if (UsbNodeGetFub.status == ERR_OK )
			{
				if(FloppyInvisible)
					LogMessage("FILE: USB device ready ");
				FloppyInvisible = FALSE;
			}
			else
			if (UsbNodeGetFub.status == asusbERR_USB_NOTFOUND)
			{
				FloppyInvisible = TRUE;
				strcpy(tmpMsg,"FILE: USB device removed ");
				brsitoa(UsbNodeGetFub.status,(UDINT)lclposstr);
				strcat(tmpMsg,lclposstr);
				LogMessage(tmpMsg);
				usbAction = USB_DEVICEUNLINK;
			}
			else
			if (UsbNodeGetFub.status != ERR_FUB_BUSY)
			{
				strcpy(tmpMsg,"FILE: Error during UsbNodeGet: ");
				brsitoa(UsbNodeGetFub.status,(UDINT)lclposstr);
				strcat(tmpMsg,lclposstr);
				LogMessage(tmpMsg);
			}
		default:
			break;
	}
}
```

### Program Logical/xml (ANSIC, version 0.00.0)
